C01845=1107.391,-76.844,-48.334,179.809,5.028,148.918
C01846=1107.386,-76.593,-48.345,179.809,5.034,148.919
C01847=1107.380,-76.344,-48.356,179.809,5.039,148.920
C01848=1107.375,-76.094,-48.367,179.809,5.044,148.922
C01849=1107.370,-75.844,-48.378,179.809,5.049,148.923
C01850=1107.365,-75.595,-48.389,179.809,5.054,148.924
C01851=1107.359,-75.345,-48.401,179.808,5.059,148.925
C01852=1107.354,-75.095,-48.411,179.808,5.064,148.926
C01853=1107.349,-74.846,-48.422,179.808,5.070,148.927
C01854=1107.344,-74.596,-48.434,179.808,5.075,148.929
C01855=1107.339,-74.346,-48.445,179.808,5.080,148.930
C01856=1107.333,-74.097,-48.456,179.808,5.085,148.931
C01857=1107.328,-73.847,-48.467,179.808,5.090,148.932
C01858=1107.323,-73.597,-48.478,179.807,5.095,148.933
C01859=1107.318,-73.383,-48.488,179.807,5.099,148.934
C01860=1107.314,-73.168,-48.497,179.808,5.104,148.935
C01861=1107.309,-72.954,-48.507,179.807,5.108,148.936
C01862=1107.305,-72.739,-48.517,179.808,5.113,148.937
C01863=1107.300,-72.525,-48.526,179.807,5.117,148.938
C01864=1107.296,-72.310,-48.536,179.807,5.122,148.939
C01865=1107.292,-72.096,-48.545,179.807,5.126,148.940
C01866=1107.287,-71.881,-48.555,179.807,5.131,148.941
C01867=1107.282,-71.631,-48.567,179.807,5.136,148.942
C01868=1107.276,-71.382,-48.578,179.807,5.141,148.943
C01869=1107.272,-71.132,-48.589,179.807,5.146,148.945
C01870=1107.266,-70.882,-48.601,179.807,5.151,148.946
C01871=1107.261,-70.632,-48.611,179.807,5.156,148.947
C01872=1107.255,-70.383,-48.623,179.807,5.161,148.948
C01873=1107.250,-70.133,-48.634,179.807,5.166,148.949
C01874=1107.246,-69.884,-48.645,179.807,5.171,148.950
C01875=1107.240,-69.634,-48.657,179.807,5.176,148.951
C01876=1107.235,-69.385,-48.668,179.807,5.181,148.952
C01877=1107.230,-69.135,-48.680,179.807,5.186,148.953
C01878=1107.225,-68.885,-48.691,179.807,5.191,148.955
C01879=1107.219,-68.635,-48.703,179.807,5.197,148.956
C01880=1107.214,-68.386,-48.713,179.807,5.201,148.957
C01881=1107.208,-68.136,-48.725,179.807,5.206,148.958
C01882=1107.204,-67.886,-48.737,179.807,5.212,148.959
C01883=1107.198,-67.636,-48.749,179.807,5.217,148.960
C01884=1107.194,-67.387,-48.760,179.808,5.222,148.961
C01885=1107.188,-67.137,-48.771,179.808,5.227,148.962
C01886=1107.183,-66.888,-48.783,179.807,5.233,148.963
C01887=1107.177,-66.638,-48.795,179.808,5.237,148.964
C01888=1107.173,-66.388,-48.806,179.808,5.242,148.966
C01889=1107.167,-66.138,-48.818,179.808,5.248,148.967
C01890=1107.163,-65.889,-48.829,179.808,5.252,148.968
C01891=1107.157,-65.639,-48.841,179.808,5.257,148.969
C01892=1107.152,-65.390,-48.852,179.808,5.262,148.970
C01893=1107.146,-65.140,-48.864,179.808,5.267,148.971
C01894=1107.142,-64.890,-48.875,179.809,5.273,148.972
C01895=1107.136,-64.640,-48.887,179.809,5.278,148.973
C01896=1107.132,-64.391,-48.898,179.809,5.283,148.974
C01897=1107.126,-64.141,-48.910,179.809,5.288,148.975
C01898=1107.120,-63.892,-48.922,179.809,5.293,148.976
C01899=1107.115,-63.642,-48.933,179.809,5.298,148.977
C01900=1107.110,-63.392,-48.945,179.809,5.303,148.978
C01901=1107.105,-63.142,-48.956,179.810,5.308,148.979
C01902=1107.100,-62.892,-48.968,179.810,5.313,148.980
C01903=1107.095,-62.643,-48.979,179.810,5.318,148.981
C01904=1107.090,-62.393,-48.991,179.810,5.322,148.982
C01905=1107.084,-62.144,-49.003,179.811,5.328,148.983
C01906=1107.079,-61.894,-49.014,179.811,5.333,148.984
C01907=1107.074,-61.645,-49.026,179.811,5.338,148.985
C01908=1107.069,-61.395,-49.038,179.812,5.343,148.986
C01909=1107.064,-61.145,-49.050,179.812,5.348,148.987
C01910=1107.058,-60.895,-49.062,179.812,5.353,148.988
C01911=1107.053,-60.645,-49.073,179.812,5.358,148.989
C01912=1107.048,-60.396,-49.085,179.813,5.362,148.990
C01913=1107.043,-60.146,-49.097,179.812,5.367,148.992
C01914=1107.038,-59.896,-49.109,179.813,5.372,148.992
C01915=1107.033,-59.682,-49.119,179.813,5.377,148.993
C01916=1107.029,-59.468,-49.130,179.813,5.381,148.994
C01917=1107.024,-59.253,-49.140,179.813,5.385,148.995
C01918=1107.020,-59.038,-49.150,179.813,5.389,148.996
C01919=1107.015,-58.825,-49.160,179.812,5.393,148.997
C01920=1107.011,-58.610,-49.170,179.812,5.397,148.998
C01921=1107.007,-58.395,-49.180,179.812,5.401,148.999
C01922=1107.002,-58.181,-49.190,179.813,5.405,149.000
C01923=1106.997,-57.931,-49.202,179.812,5.409,149.001
C01924=1106.992,-57.682,-49.213,179.812,5.414,149.002
C01925=1106.987,-57.433,-49.226,179.812,5.418,149.003
C01926=1106.981,-57.183,-49.238,179.812,5.423,149.004
C01927=1106.977,-56.933,-49.249,179.812,5.428,149.005
C01928=1106.971,-56.683,-49.261,179.812,5.433,149.006
C01929=1106.966,-56.434,-49.274,179.811,5.438,149.007
C01930=1106.961,-56.184,-49.286,179.812,5.442,149.008
C01931=1106.956,-55.934,-49.297,179.811,5.447,149.009
C01932=1106.951,-55.685,-49.310,179.811,5.452,149.010
C01933=1106.946,-55.435,-49.321,179.812,5.457,149.011
C01934=1106.940,-55.185,-49.333,179.811,5.461,149.013
C01935=1106.935,-54.936,-49.346,179.811,5.466,149.013
C01936=1106.930,-54.686,-49.357,179.811,5.471,149.015
C01937=1106.925,-54.437,-49.370,179.810,5.475,149.016
C01938=1106.920,-54.187,-49.382,179.811,5.480,149.017
C01939=1106.914,-53.937,-49.394,179.811,5.485,149.018
C01940=1106.909,-53.688,-49.406,179.810,5.489,149.019
C01941=1106.905,-53.438,-49.417,179.810,5.494,149.020
C01942=1106.900,-53.187,-49.430,179.810,5.499,149.021
C01943=1106.895,-52.938,-49.442,179.810,5.504,149.022
C01944=1106.889,-52.688,-49.454,179.810,5.508,149.023
C01945=1106.884,-52.439,-49.467,179.809,5.513,149.024
C01946=1106.879,-52.189,-49.479,179.809,5.518,149.025
C01947=1106.874,-51.940,-49.491,179.810,5.522,149.026
C01948=1106.869,-51.690,-49.503,179.809,5.527,149.028
C01949=1106.864,-51.440,-49.515,179.809,5.532,149.029
C01950=1106.858,-51.191,-49.527,179.809,5.537,149.030
C01951=1106.853,-50.941,-49.539,179.809,5.541,149.031
C01952=1106.848,-50.691,-49.552,179.809,5.546,149.032
C01953=1106.842,-50.441,-49.563,179.809,5.551,149.033
C01954=1106.837,-50.192,-49.576,179.808,5.555,149.034
C01955=1106.832,-49.942,-49.588,179.808,5.560,149.035
C01956=1106.827,-49.693,-49.600,179.809,5.565,149.036
C01957=1106.822,-49.444,-49.612,179.808,5.569,149.037
C01958=1106.817,-49.193,-49.625,179.808,5.574,149.038
C01959=1106.812,-48.944,-49.637,179.808,5.578,149.039
C01960=1106.807,-48.694,-49.649,179.808,5.584,149.040
C01961=1106.802,-48.445,-49.662,179.808,5.589,149.042
C01962=1106.796,-48.195,-49.674,179.807,5.593,149.043
C01963=1106.791,-47.945,-49.686,179.807,5.598,149.044
C01964=1106.786,-47.695,-49.698,179.807,5.603,149.045
C01965=1106.781,-47.446,-49.711,179.807,5.607,149.046
C01966=1106.775,-47.197,-49.723,179.807,5.612,149.047
C01967=1106.770,-46.947,-49.735,179.807,5.617,149.048
C01968=1106.765,-46.697,-49.748,179.806,5.621,149.049
C01969=1106.760,-46.447,-49.760,179.806,5.627,149.050
C01970=1106.755,-46.198,-49.773,179.806,5.630,149.051
C01971=1106.751,-45.983,-49.783,179.807,5.635,149.052
C01972=1106.747,-45.768,-49.793,179.806,5.639,149.053
C01973=1106.741,-45.555,-49.804,179.806,5.643,149.054
C01974=1106.737,-45.340,-49.815,179.806,5.647,149.055
C01975=1106.733,-45.126,-49.826,179.805,5.651,149.056
C01976=1106.729,-44.911,-49.836,179.805,5.655,149.057
C01977=1106.724,-44.697,-49.847,179.805,5.659,149.058
C01978=1106.720,-44.482,-49.858,179.805,5.663,149.059
C01979=1106.715,-44.233,-49.871,179.805,5.668,149.060
C01980=1106.709,-43.983,-49.882,179.805,5.673,149.061
C01981=1106.704,-43.734,-49.895,179.805,5.677,149.062
C01982=1106.699,-43.485,-49.908,179.805,5.682,149.063
C01983=1106.694,-43.235,-49.920,179.804,5.686,149.064
C01984=1106.689,-42.985,-49.932,179.804,5.692,149.065
C01985=1106.684,-42.735,-49.945,179.804,5.697,149.066
C01986=1106.679,-42.486,-49.958,179.805,5.701,149.067
C01987=1106.674,-42.236,-49.970,179.805,5.706,149.068
C01988=1106.668,-41.986,-49.983,179.805,5.711,149.069
C01989=1106.663,-41.736,-49.996,179.806,5.716,149.070
C01990=1106.658,-41.487,-50.008,179.806,5.721,149.071
C01991=1106.653,-41.238,-50.021,179.806,5.726,149.072
C01992=1106.647,-40.988,-50.033,179.806,5.731,149.073
C01993=1106.642,-40.739,-50.045,179.807,5.735,149.074
C01994=1106.638,-40.488,-50.058,179.807,5.740,149.075
C01995=1106.633,-40.239,-50.071,179.808,5.745,149.076
C01996=1106.628,-39.990,-50.084,179.808,5.750,149.077
C01997=1106.621,-39.740,-50.096,179.808,5.755,149.078
C01998=1106.617,-39.490,-50.109,179.809,5.759,149.079
C01999=1106.612,-39.240,-50.122,179.809,5.764,149.080
C02000=1106.607,-38.991,-50.134,179.809,5.769,149.081
C02001=1106.602,-38.742,-50.147,179.810,5.774,149.082
C02002=1106.597,-38.492,-50.160,179.810,5.778,149.083
C02003=1106.591,-38.242,-50.173,179.811,5.783,149.084
C02004=1106.586,-37.993,-50.186,179.811,5.788,149.084
C02005=1106.581,-37.743,-50.197,179.811,5.792,149.085
C02006=1106.576,-37.493,-50.210,179.811,5.796,149.086
C02007=1106.571,-37.243,-50.223,179.812,5.801,149.087
C02008=1106.565,-36.994,-50.236,179.812,5.806,149.088
C02009=1106.560,-36.744,-50.249,179.813,5.811,149.089
C02010=1106.555,-36.494,-50.262,179.814,5.815,149.090
C02011=1106.550,-36.245,-50.274,179.814,5.819,149.091
C02012=1106.544,-35.995,-50.288,179.814,5.824,149.091
C02013=1106.540,-35.745,-50.301,179.815,5.828,149.092
C02014=1106.535,-35.496,-50.313,179.815,5.833,149.093
C02015=1106.530,-35.247,-50.326,179.815,5.837,149.094
C02016=1106.524,-34.996,-50.339,179.815,5.842,149.095
C02017=1106.519,-34.747,-50.352,179.816,5.847,149.096
C02018=1106.514,-34.498,-50.364,179.816,5.851,149.097
C02019=1106.510,-34.248,-50.377,179.816,5.855,149.098
C02020=1106.504,-33.998,-50.391,179.817,5.860,149.099
C02021=1106.499,-33.749,-50.403,179.817,5.864,149.099
C02022=1106.494,-33.499,-50.416,179.817,5.868,149.100
C02023=1106.488,-33.249,-50.429,179.818,5.873,149.101
C02024=1106.483,-33.000,-50.442,179.818,5.878,149.102
C02025=1106.479,-32.750,-50.455,179.819,5.882,149.103
C02026=1106.474,-32.501,-50.468,179.818,5.886,149.104
C02027=1106.469,-32.287,-50.480,179.819,5.890,149.105
C02028=1106.464,-32.072,-50.491,179.820,5.894,149.105
C02029=1106.460,-31.858,-50.502,179.820,5.898,149.106
C02030=1106.455,-31.643,-50.513,179.820,5.902,149.107
C02031=1106.452,-31.430,-50.524,179.820,5.906,149.108
C02032=1106.447,-31.215,-50.536,179.820,5.909,149.109
C02033=1106.443,-31.001,-50.546,179.821,5.913,149.109
C02034=1106.438,-30.786,-50.558,179.820,5.917,149.110
C02035=1106.433,-30.537,-50.570,179.821,5.921,149.111
C02036=1106.428,-30.287,-50.584,179.821,5.926,149.112
C02037=1106.423,-30.038,-50.597,179.821,5.930,149.113
C02038=1106.418,-29.788,-50.610,179.822,5.935,149.114
C02039=1106.413,-29.538,-50.623,179.822,5.940,149.115
C02040=1106.407,-29.289,-50.636,179.822,5.944,149.116
C02041=1106.402,-29.039,-50.650,179.822,5.948,149.116
C02042=1106.397,-28.790,-50.663,179.822,5.952,149.117
C02043=1106.393,-28.540,-50.676,179.823,5.957,149.118
C02044=1106.387,-28.290,-50.689,179.823,5.962,149.119
C02045=1106.382,-28.041,-50.702,179.823,5.966,149.120
C02046=1106.377,-27.791,-50.716,179.824,5.970,149.121
C02047=1106.372,-27.542,-50.729,179.824,5.975,149.122
C02048=1106.367,-27.292,-50.741,179.823,5.979,149.123
C02049=1106.361,-27.042,-50.755,179.824,5.984,149.124
C02050=1106.357,-26.793,-50.768,179.824,5.989,149.125
C02051=1106.351,-26.543,-50.782,179.824,5.993,149.126
C02052=1106.347,-26.293,-50.795,179.824,5.998,149.127
C02053=1106.341,-26.044,-50.808,179.824,6.002,149.128
C02054=1106.337,-25.794,-50.821,179.825,6.007,149.129
C02055=1106.331,-25.545,-50.835,179.824,6.012,149.130
C02056=1106.327,-25.295,-50.848,179.825,6.016,149.131
C02057=1106.321,-25.046,-50.861,179.825,6.021,149.132
C02058=1106.316,-24.796,-50.874,179.825,6.025,149.133
C02059=1106.311,-24.547,-50.888,179.826,6.030,149.133
C02060=1106.306,-24.297,-50.901,179.826,6.035,149.135
C02061=1106.300,-24.047,-50.915,179.826,6.040,149.136
C02062=1106.296,-23.798,-50.928,179.827,6.044,149.136
C02063=1106.290,-23.548,-50.941,179.827,6.049,149.137
C02064=1106.285,-23.299,-50.955,179.828,6.054,149.138
C02065=1106.280,-23.049,-50.968,179.828,6.058,149.139
C02066=1106.275,-22.800,-50.981,179.828,6.063,149.140
C02067=1106.270,-22.550,-50.995,179.828,6.068,149.141
C02068=1106.264,-22.300,-51.008,179.829,6.072,149.142
C02069=1106.260,-22.051,-51.022,179.829,6.077,149.143
C02070=1106.254,-21.801,-51.035,179.829,6.082,149.144
C02071=1106.250,-21.552,-51.049,179.830,6.086,149.145
C02072=1106.245,-21.302,-51.062,179.830,6.091,149.146
C02073=1106.240,-21.053,-51.076,179.830,6.095,149.147
C02074=1106.235,-20.802,-51.089,179.831,6.100,149.147
C02075=1106.229,-20.553,-51.103,179.831,6.105,149.148
C02076=1106.225,-20.303,-51.116,179.832,6.109,149.149
C02077=1106.219,-20.054,-51.130,179.832,6.114,149.150
C02078=1106.214,-19.804,-51.144,179.833,6.119,149.151
C02079=1106.209,-19.555,-51.157,179.833,6.123,149.152
C02080=1106.204,-19.305,-51.171,179.833,6.127,149.153
C02081=1106.199,-19.056,-51.184,179.834,6.132,149.154
C02082=1106.194,-18.806,-51.197,179.834,6.137,149.155
C02083=1106.189,-18.592,-51.209,179.834,6.141,149.156
C02084=1106.185,-18.378,-51.222,179.835,6.145,149.156
C02085=1106.180,-18.163,-51.233,179.835,6.149,149.157
C02086=1106.177,-17.949,-51.245,179.835,6.153,149.158
C02087=1106.172,-17.735,-51.256,179.836,6.157,149.159
C02088=1106.168,-17.521,-51.268,179.836,6.161,149.159
C02089=1106.163,-17.307,-51.280,179.836,6.164,149.160
C02090=1106.158,-17.092,-51.291,179.837,6.168,149.161
C02091=1106.154,-16.843,-51.305,179.837,6.173,149.162
C02092=1106.149,-16.594,-51.319,179.838,6.177,149.163
C02093=1106.143,-16.344,-51.332,179.838,6.182,149.163
C02094=1106.138,-16.094,-51.347,179.839,6.187,149.164
C02095=1106.133,-15.845,-51.360,179.839,6.192,149.165
C02096=1106.128,-15.595,-51.374,179.839,6.195,149.166
C02097=1106.123,-15.345,-51.388,179.840,6.200,149.167
C02098=1106.118,-15.096,-51.401,179.840,6.205,149.168
C02099=1106.113,-14.846,-51.415,179.841,6.209,149.169
C02100=1106.108,-14.596,-51.429,179.842,6.214,149.170
C02101=1106.103,-14.347,-51.443,179.842,6.219,149.170
C02102=1106.098,-14.098,-51.457,179.843,6.223,149.171
C02103=1106.093,-13.848,-51.470,179.842,6.227,149.172
C02104=1106.088,-13.599,-51.484,179.843,6.232,149.173
C02105=1106.083,-13.349,-51.498,179.843,6.237,149.174
C02106=1106.078,-13.099,-51.513,179.844,6.241,149.175
C02107=1106.073,-12.850,-51.525,179.845,6.246,149.176
C02108=1106.068,-12.600,-51.540,179.845,6.251,149.176
C02109=1106.063,-12.351,-51.554,179.845,6.254,149.177
C02110=1106.057,-12.102,-51.568,179.846,6.259,149.178
C02111=1106.052,-11.852,-51.582,179.847,6.264,149.179
C02112=1106.047,-11.602,-51.596,179.847,6.268,149.180
C02113=1106.043,-11.352,-51.609,179.848,6.273,149.181
C02114=1106.037,-11.103,-51.623,179.848,6.278,149.182
C02115=1106.032,-10.853,-51.637,179.849,6.282,149.183
C02116=1106.027,-10.604,-51.652,179.849,6.286,149.183
C02117=1106.022,-10.355,-51.666,179.850,6.291,149.184
C02118=1106.017,-10.105,-51.680,179.850,6.295,149.185
C02119=1106.013,-9.856,-51.694,179.851,6.300,149.186
C02120=1106.008,-9.606,-51.708,179.851,6.305,149.187
C02121=1106.002,-9.356,-51.721,179.852,6.309,149.187
C02122=1105.997,-9.106,-51.735,179.853,6.314,149.188
C02123=1105.992,-8.857,-51.750,179.853,6.318,149.189
C02124=1105.987,-8.607,-51.764,179.853,6.322,149.190
C02125=1105.981,-8.358,-51.778,179.854,6.327,149.191
C02126=1105.976,-8.108,-51.792,179.855,6.332,149.192
C02127=1105.971,-7.859,-51.806,179.855,6.336,149.193
C02128=1105.966,-7.609,-51.821,179.856,6.341,149.194
C02129=1105.961,-7.359,-51.835,179.857,6.345,149.194
C02130=1105.956,-7.110,-51.849,179.857,6.349,149.195
C02131=1105.951,-6.860,-51.863,179.857,6.354,149.196
C02132=1105.947,-6.611,-51.877,179.858,6.359,149.197
C02133=1105.942,-6.361,-51.891,179.859,6.363,149.198
C02134=1105.937,-6.112,-51.905,179.859,6.368,149.198
C02135=1105.931,-5.863,-51.919,179.860,6.372,149.199
C02136=1105.926,-5.613,-51.934,179.861,6.377,149.200
C02137=1105.921,-5.363,-51.948,179.861,6.381,149.201
C02138=1105.916,-5.114,-51.962,179.861,6.385,149.202
C02139=1105.912,-4.900,-51.974,179.862,6.390,149.202
C02140=1105.907,-4.686,-51.987,179.862,6.393,149.203
C02141=1105.903,-4.471,-52.000,179.863,6.397,149.204
C02142=1105.899,-4.257,-52.012,179.863,6.402,149.205
C02143=1105.894,-4.044,-52.024,179.864,6.405,149.205
C02144=1105.890,-3.829,-52.036,179.864,6.409,149.206
C02145=1105.886,-3.615,-52.048,179.865,6.413,149.207
C02146=1105.881,-3.401,-52.060,179.865,6.416,149.207
C02147=1105.877,-3.151,-52.075,179.866,6.421,149.208
C02148=1105.872,-2.902,-52.089,179.867,6.426,149.209
C02149=1105.867,-2.653,-52.104,179.867,6.431,149.210
C02150=1105.861,-2.402,-52.119,179.868,6.435,149.211
C02151=1105.856,-2.153,-52.133,179.869,6.440,149.212
C02152=1105.851,-1.904,-52.147,179.869,6.444,149.212
C02153=1105.846,-1.654,-52.161,179.869,6.448,149.213
C02154=1105.841,-1.405,-52.176,179.870,6.453,149.214
C02155=1105.836,-1.155,-52.191,179.871,6.457,149.215
C02156=1105.831,-0.906,-52.205,179.871,6.462,149.216
C02157=1105.826,-0.656,-52.219,179.872,6.466,149.217
C02158=1105.821,-0.406,-52.233,179.873,6.471,149.217
C02159=1105.816,-0.157,-52.249,179.873,6.476,149.218
C02160=1105.811,0.093,-52.263,179.874,6.480,149.219
C02161=1105.805,0.342,-52.277,179.875,6.485,149.220
C02162=1105.801,0.591,-52.292,179.875,6.490,149.221
C02163=1105.796,0.841,-52.306,179.876,6.494,149.221
C02164=1105.791,1.091,-52.321,179.877,6.499,149.222
C02165=1105.786,1.340,-52.335,179.877,6.503,149.223
C02166=1105.780,1.590,-52.351,179.878,6.508,149.224
C02167=1105.776,1.839,-52.365,179.878,6.512,149.225
C02168=1105.771,2.089,-52.379,179.879,6.516,149.226
C02169=1105.766,2.338,-52.394,179.879,6.521,149.227
C02170=1105.761,2.588,-52.408,179.880,6.525,149.227
C02171=1105.756,2.837,-52.424,179.881,6.530,149.228
C02172=1105.751,3.087,-52.438,179.881,6.535,149.229
C02173=1105.746,3.337,-52.453,179.882,6.539,149.230
C02174=1105.741,3.586,-52.468,179.883,6.544,149.231
C02175=1105.735,3.836,-52.482,179.883,6.548,149.231
C02176=1105.731,4.085,-52.497,179.884,6.553,149.232
C02177=1105.726,4.335,-52.512,179.884,6.558,149.233
C02178=1105.721,4.584,-52.526,179.885,6.562,149.234
C02179=1105.715,4.834,-52.542,179.886,6.567,149.235
C02180=1105.710,5.083,-52.556,179.887,6.572,149.236
C02181=1105.706,5.333,-52.571,179.887,6.576,149.237
C02182=1105.701,5.582,-52.585,179.888,6.581,149.237
C02183=1105.695,5.832,-52.601,179.889,6.585,149.238
C02184=1105.690,6.081,-52.615,179.889,6.590,149.239
C02185=1105.686,6.330,-52.630,179.890,6.595,149.240
C02186=1105.680,6.580,-52.645,179.891,6.599,149.241
C02187=1105.675,6.830,-52.660,179.891,6.604,149.241
C02188=1105.671,7.079,-52.674,179.892,6.608,149.242
C02189=1105.665,7.329,-52.690,179.892,6.613,149.243
C02190=1105.661,7.578,-52.705,179.893,6.618,149.244
C02191=1105.656,7.827,-52.719,179.894,6.622,149.245
C02192=1105.650,8.077,-52.735,179.894,6.627,149.246
C02193=1105.645,8.327,-52.749,179.895,6.632,149.247
C02194=1105.641,8.576,-52.764,179.896,6.636,149.247
C02195=1105.636,8.791,-52.777,179.896,6.640,149.248
C02196=1105.632,9.004,-52.790,179.897,6.644,149.249
C02197=1105.628,9.218,-52.803,179.897,6.648,149.250
C02198=1105.623,9.432,-52.815,179.897,6.652,149.250
C02199=1105.619,9.646,-52.828,179.897,6.656,149.251
C02200=1105.614,9.860,-52.841,179.898,6.659,149.252
C02201=1105.611,10.074,-52.854,179.899,6.663,149.253
C02202=1105.606,10.288,-52.867,179.899,6.667,149.253
C02203=1105.601,10.538,-52.882,179.899,6.671,149.254
C02204=1105.595,10.787,-52.897,179.899,6.676,149.255
C02205=1105.591,11.036,-52.912,179.900,6.681,149.256
C02206=1105.586,11.286,-52.927,179.901,6.685,149.257
C02207=1105.581,11.536,-52.943,179.901,6.689,149.258
C02208=1105.576,11.785,-52.958,179.901,6.694,149.259
C02209=1105.571,12.035,-52.972,179.902,6.698,149.259
C02210=1105.566,12.284,-52.987,179.902,6.702,149.260
C02211=1105.561,12.534,-53.003,179.902,6.707,149.261
C02212=1105.556,12.783,-53.018,179.903,6.712,149.262
C02213=1105.550,13.033,-53.033,179.903,6.716,149.263
C02214=1105.546,13.282,-53.048,179.904,6.720,149.264
C02215=1105.541,13.532,-53.064,179.904,6.725,149.264
C02216=1105.536,13.781,-53.079,179.905,6.729,149.265
C02217=1105.531,14.031,-53.094,179.905,6.733,149.266
C02218=1105.526,14.280,-53.109,179.905,6.738,149.267
C02219=1105.521,14.530,-53.124,179.906,6.742,149.268
C02220=1105.516,14.779,-53.139,179.907,6.747,149.269
C02221=1105.511,15.029,-53.155,179.907,6.751,149.270
C02222=1105.506,15.278,-53.170,179.907,6.755,149.270
C02223=1105.501,15.528,-53.185,179.909,6.760,149.271
C02224=1105.496,15.777,-53.200,179.908,6.764,149.272
C02225=1105.491,16.026,-53.216,179.909,6.768,149.273
C02226=1105.487,16.276,-53.231,179.910,6.773,149.274
C02227=1105.481,16.526,-53.247,179.910,6.777,149.274
C02228=1105.476,16.775,-53.262,179.911,6.781,149.275
C02229=1105.471,17.024,-53.277,179.911,6.786,149.276
C02230=1105.466,17.273,-53.293,179.912,6.790,149.277
C02231=1105.462,17.524,-53.307,179.912,6.794,149.278
C02232=1105.456,17.773,-53.323,179.913,6.799,149.279
C02233=1105.451,18.023,-53.339,179.914,6.803,149.279
C02234=1105.446,18.272,-53.354,179.914,6.807,149.280
C02235=1105.441,18.521,-53.369,179.914,6.812,149.281
C02236=1105.437,18.771,-53.385,179.915,6.816,149.282
C02237=1105.431,19.020,-53.400,179.915,6.820,149.283
C02238=1105.426,19.270,-53.416,179.916,6.824,149.283
C02239=1105.421,19.519,-53.431,179.917,6.829,149.284
C02240=1105.416,19.769,-53.447,179.917,6.833,149.285
C02241=1105.411,20.018,-53.462,179.918,6.837,149.286
C02242=1105.406,20.267,-53.477,179.918,6.842,149.287
C02243=1105.401,20.517,-53.493,179.919,6.846,149.287
C02244=1105.396,20.767,-53.509,179.919,6.850,149.288
C02245=1105.392,21.016,-53.524,179.920,6.855,149.289
C02246=1105.386,21.265,-53.539,179.921,6.859,149.290
C02247=1105.381,21.516,-53.555,179.921,6.863,149.290
C02248=1105.377,21.765,-53.570,179.922,6.868,149.291
C02249=1105.371,22.014,-53.586,179.923,6.872,149.292
C02250=1105.366,22.263,-53.602,179.923,6.876,149.293
C02251=1105.362,22.477,-53.616,179.924,6.880,149.293
C02252=1105.358,22.691,-53.629,179.925,6.884,149.294
C02253=1105.354,22.905,-53.642,179.925,6.887,149.295
C02254=1105.349,23.119,-53.656,179.925,6.891,149.295
C02255=1105.346,23.333,-53.669,179.926,6.894,149.296
C02256=1105.341,23.547,-53.683,179.926,6.898,149.297
C02257=1105.337,23.761,-53.696,179.927,6.902,149.297
C02258=1105.332,23.974,-53.709,179.928,6.905,149.298
C02259=1105.328,24.224,-53.725,179.928,6.909,149.299
C02260=1105.322,24.474,-53.741,179.929,6.914,149.300
C02261=1105.317,24.723,-53.756,179.930,6.918,149.300
C02262=1105.313,24.972,-53.772,179.930,6.922,149.301
C02263=1105.308,25.222,-53.788,179.931,6.926,149.302
C02264=1105.302,25.471,-53.803,179.932,6.931,149.302
C02265=1105.298,25.721,-53.819,179.932,6.935,149.303
C02266=1105.292,25.971,-53.835,179.933,6.939,149.304
C02267=1105.288,26.219,-53.851,179.934,6.943,149.305
C02268=1105.283,26.469,-53.867,179.934,6.948,149.306
C02269=1105.278,26.719,-53.882,179.935,6.951,149.306
C02270=1105.273,26.969,-53.898,179.936,6.956,149.307
C02271=1105.268,27.218,-53.914,179.937,6.960,149.308
C02272=1105.262,27.467,-53.930,179.937,6.964,149.308
C02273=1105.258,27.717,-53.945,179.938,6.968,149.309
C02274=1105.253,27.966,-53.961,179.939,6.973,149.310
C02275=1105.248,28.215,-53.977,179.939,6.976,149.311
C02276=1105.243,28.465,-53.993,179.940,6.981,149.311
C02277=1105.238,28.715,-54.009,179.941,6.985,149.312
C02278=1105.233,28.964,-54.025,179.942,6.990,149.313
C02279=1105.228,29.213,-54.041,179.942,6.993,149.313
C02280=1105.223,29.464,-54.057,179.943,6.997,149.314
C02281=1105.219,29.712,-54.073,179.944,7.002,149.315
C02282=1105.213,29.961,-54.088,179.944,7.006,149.316
C02283=1105.209,30.211,-54.105,179.945,7.010,149.316
C02284=1105.203,30.460,-54.121,179.946,7.014,149.317
C02285=1105.199,30.710,-54.136,179.946,7.018,149.318
C02286=1105.194,30.959,-54.153,179.947,7.023,149.318
C02287=1105.189,31.209,-54.169,179.949,7.027,149.319
C02288=1105.184,31.458,-54.185,179.949,7.030,149.320
C02289=1105.178,31.707,-54.201,179.950,7.035,149.320
C02290=1105.174,31.958,-54.217,179.951,7.039,149.321
C02291=1105.168,32.206,-54.233,179.952,7.044,149.322
C02292=1105.164,32.456,-54.249,179.952,7.047,149.323
C02293=1105.159,32.705,-54.265,179.953,7.051,149.323
C02294=1105.154,32.955,-54.281,179.954,7.056,149.324
C02295=1105.149,33.204,-54.297,179.955,7.059,149.325
C02296=1105.144,33.454,-54.313,179.956,7.064,149.325
C02297=1105.139,33.703,-54.330,179.956,7.068,149.326
C02298=1105.134,33.953,-54.346,179.957,7.072,149.327
C02299=1105.129,34.202,-54.362,179.958,7.076,149.327
C02300=1105.124,34.452,-54.378,179.959,7.080,149.328
C02301=1105.119,34.701,-54.394,179.959,7.084,149.329
C02302=1105.114,34.951,-54.410,179.960,7.088,149.329
C02303=1105.109,35.200,-54.426,179.961,7.093,149.330
C02304=1105.105,35.449,-54.443,179.963,7.097,149.331
C02305=1105.099,35.699,-54.459,179.963,7.100,149.331
C02306=1105.095,35.948,-54.475,179.964,7.105,149.332
C02307=1105.090,36.162,-54.489,179.965,7.108,149.333
C02308=1105.086,36.375,-54.503,179.965,7.112,149.333
C02309=1105.082,36.590,-54.517,179.966,7.115,149.334
C02310=1105.078,36.803,-54.531,179.967,7.119,149.334
C02311=1105.073,37.018,-54.545,179.967,7.123,149.335
C02312=1105.069,37.231,-54.559,179.968,7.126,149.336
C02313=1105.065,37.445,-54.573,179.969,7.129,149.336
C02314=1105.061,37.659,-54.587,179.970,7.132,149.337
C02315=1105.056,37.908,-54.604,179.971,7.137,149.337
C02316=1105.051,38.158,-54.619,179.972,7.141,149.338
C02317=1105.046,38.407,-54.636,179.972,7.145,149.339
C02318=1105.040,38.656,-54.653,179.973,7.149,149.339
C02319=1105.036,38.906,-54.669,179.974,7.153,149.340
C02320=1105.031,39.155,-54.685,179.975,7.157,149.341
C02321=1105.026,39.405,-54.702,179.976,7.161,149.341
C02322=1105.021,39.655,-54.718,179.977,7.165,149.342
C02323=1105.016,39.903,-54.734,179.978,7.170,149.343
C02324=1105.011,40.153,-54.751,179.979,7.173,149.343
C02325=1105.006,40.402,-54.768,179.980,7.177,149.344
C02326=1105.001,40.651,-54.784,179.981,7.182,149.345
C02327=1104.997,40.902,-54.800,179.982,7.186,149.345
C02328=1104.992,41.150,-54.817,179.982,7.190,149.346
C02329=1104.986,41.400,-54.834,179.983,7.194,149.346
C02330=1104.981,41.649,-54.850,179.984,7.198,149.347
C02331=1104.977,41.898,-54.867,179.985,7.202,149.348
C02332=1104.972,42.149,-54.883,179.986,7.206,149.348
C02333=1104.967,42.397,-54.899,179.987,7.210,149.349
C02334=1104.962,42.647,-54.916,179.988,7.213,149.350
C02335=1104.957,42.897,-54.933,179.989,7.218,149.350
C02336=1104.952,43.145,-54.949,179.990,7.222,149.351
C02337=1104.948,43.395,-54.966,179.991,7.226,149.352
C02338=1104.942,43.645,-54.983,179.992,7.230,149.352
C02339=1104.937,43.894,-54.999,179.993,7.234,149.353
C02340=1104.933,44.144,-55.016,179.994,7.238,149.353
C02341=1104.927,44.393,-55.033,179.995,7.242,149.354
C02342=1104.922,44.642,-55.049,179.996,7.246,149.355
C02343=1104.918,44.892,-55.066,179.997,7.250,149.355
C02344=1104.913,45.141,-55.083,179.998,7.254,149.356
C02345=1104.907,45.390,-55.099,179.998,7.258,149.357
C02346=1104.903,45.640,-55.116,180.000,7.262,149.357
C02347=1104.899,45.889,-55.133,-179.999,7.266,149.358
C02348=1104.893,46.138,-55.150,-179.998,7.270,149.358
C02349=1104.888,46.388,-55.166,-179.997,7.274,149.359
C02350=1104.883,46.638,-55.184,-179.996,7.278,149.360
C02351=1104.879,46.887,-55.200,-179.995,7.282,149.360
C02352=1104.873,47.136,-55.217,-179.994,7.286,149.361
C02353=1104.868,47.386,-55.234,-179.993,7.290,149.361
C02354=1104.864,47.635,-55.250,-179.992,7.294,149.362
C02355=1104.859,47.885,-55.267,-179.991,7.298,149.362
C02356=1104.853,48.134,-55.284,-179.990,7.302,149.363
C02357=1104.849,48.383,-55.301,-179.989,7.306,149.364
C02358=1104.844,48.633,-55.318,-179.988,7.310,149.364
C02359=1104.840,48.882,-55.335,-179.986,7.314,149.365
C02360=1104.835,49.131,-55.352,-179.986,7.318,149.365
C02361=1104.829,49.380,-55.369,-179.985,7.322,149.366
C02362=1104.825,49.630,-55.386,-179.983,7.326,149.367
C02363=1104.821,49.844,-55.400,-179.983,7.329,149.367
C02364=1104.816,50.058,-55.415,-179.982,7.333,149.368
C02365=1104.812,50.271,-55.429,-179.981,7.336,149.368
C02366=1104.808,50.485,-55.444,-179.980,7.340,149.369
C02367=1104.804,50.699,-55.458,-179.979,7.343,149.369
C02368=1104.799,50.913,-55.473,-179.978,7.346,149.370
C02369=1104.795,51.126,-55.488,-179.978,7.350,149.370
C02370=1104.791,51.340,-55.502,-179.977,7.353,149.371
C02371=1104.786,51.589,-55.519,-179.976,7.357,149.371
C02372=1104.781,51.839,-55.536,-179.974,7.361,149.372
C02373=1104.776,52.088,-55.553,-179.973,7.365,149.372
C02374=1104.772,52.337,-55.570,-179.973,7.369,149.373
C02375=1104.767,52.587,-55.588,-179.971,7.373,149.374
C02376=1104.761,52.836,-55.604,-179.970,7.377,149.374
C02377=1104.756,53.086,-55.621,-179.969,7.381,149.375
C02378=1104.752,53.335,-55.639,-179.968,7.385,149.375
C02379=1104.747,53.584,-55.656,-179.967,7.389,149.376
C02380=1104.742,53.834,-55.673,-179.965,7.393,149.376
C02381=1104.737,54.083,-55.691,-179.964,7.397,149.377
C02382=1104.732,54.332,-55.707,-179.964,7.401,149.378
C02383=1104.727,54.582,-55.724,-179.962,7.404,149.378
C02384=1104.722,54.831,-55.742,-179.961,7.409,149.379
C02385=1104.718,55.080,-55.759,-179.960,7.413,149.379
C02386=1104.713,55.330,-55.776,-179.958,7.417,149.380
C02387=1104.708,55.579,-55.794,-179.958,7.420,149.381
C02388=1104.703,55.829,-55.811,-179.956,7.424,149.381
C02389=1104.698,56.078,-55.828,-179.955,7.429,149.382
C02390=1104.693,56.327,-55.845,-179.954,7.433,149.382
C02391=1104.688,56.576,-55.862,-179.953,7.436,149.383
C02392=1104.683,56.826,-55.880,-179.952,7.440,149.383
C02393=1104.679,57.075,-55.897,-179.951,7.444,149.384
C02394=1104.673,57.325,-55.914,-179.949,7.449,149.384
C02395=1104.668,57.574,-55.932,-179.949,7.452,149.385
C02396=1104.664,57.824,-55.949,-179.947,7.456,149.386
C02397=1104.659,58.073,-55.967,-179.946,7.460,149.386
C02398=1104.654,58.323,-55.984,-179.945,7.464,149.387
C02399=1104.650,58.571,-56.001,-179.943,7.468,149.387
C02400=1104.644,58.821,-56.019,-179.943,7.472,149.388
C02401=1104.639,59.070,-56.036,-179.941,7.476,149.388
C02402=1104.634,59.319,-56.053,-179.940,7.480,149.389
C02403=1104.630,59.568,-56.071,-179.939,7.484,149.389
C02404=1104.624,59.818,-56.088,-179.938,7.487,149.390
C02405=1104.619,60.067,-56.106,-179.937,7.491,149.391
C02406=1104.615,60.317,-56.123,-179.935,7.495,149.391
C02407=1104.610,60.566,-56.141,-179.934,7.500,149.392
C02408=1104.605,60.815,-56.159,-179.933,7.504,149.392
C02409=1104.600,61.065,-56.176,-179.932,7.507,149.393
C02410=1104.596,61.314,-56.193,-179.931,7.511,149.393
C02411=1104.590,61.564,-56.211,-179.929,7.515,149.394
C02412=1104.586,61.813,-56.229,-179.928,7.519,149.394
C02413=1104.581,62.062,-56.247,-179.926,7.523,149.395
C02414=1104.576,62.311,-56.263,-179.926,7.527,149.395
C02415=1104.571,62.561,-56.281,-179.924,7.531,149.396
C02416=1104.566,62.810,-56.299,-179.923,7.535,149.396
C02417=1104.561,63.060,-56.317,-179.922,7.539,149.397
C02418=1104.556,63.309,-56.335,-179.921,7.543,149.398
C02419=1104.552,63.522,-56.349,-179.920,7.546,149.398
C02420=1104.548,63.736,-56.365,-179.919,7.549,149.398
C02421=1104.544,63.950,-56.379,-179.918,7.552,149.399
C02422=1104.540,64.164,-56.395,-179.916,7.556,149.399
C02423=1104.536,64.377,-56.410,-179.915,7.559,149.400
C02424=1104.532,64.591,-56.425,-179.914,7.563,149.400
C02425=1104.527,64.805,-56.440,-179.913,7.566,149.401
C02426=1104.523,65.018,-56.456,-179.912,7.570,149.401
C02427=1104.518,65.267,-56.473,-179.911,7.574,149.402
C02428=1104.514,65.517,-56.492,-179.910,7.577,149.402
C02429=1104.509,65.767,-56.509,-179.909,7.581,149.403
C02430=1104.504,66.016,-56.527,-179.907,7.585,149.403
C02431=1104.499,66.265,-56.545,-179.906,7.589,149.404
C02432=1104.495,66.514,-56.562,-179.904,7.593,149.404
C02433=1104.490,66.763,-56.580,-179.903,7.597,149.405
C02434=1104.485,67.013,-56.598,-179.902,7.601,149.405
C02435=1104.480,67.262,-56.616,-179.901,7.605,149.406
C02436=1104.475,67.511,-56.634,-179.900,7.609,149.406
C02437=1104.470,67.760,-56.652,-179.898,7.613,149.407
C02438=1104.465,68.010,-56.670,-179.897,7.617,149.407
C02439=1104.461,68.259,-56.688,-179.895,7.621,149.408
C02440=1104.456,68.509,-56.706,-179.894,7.625,149.408
C02441=1104.451,68.758,-56.724,-179.893,7.628,149.409
C02442=1104.446,69.007,-56.742,-179.892,7.632,149.410
C02443=1104.441,69.257,-56.759,-179.890,7.636,149.410
C02444=1104.436,69.506,-56.777,-179.889,7.640,149.410
C02445=1104.431,69.755,-56.795,-179.888,7.644,149.411
C02446=1104.426,70.004,-56.813,-179.886,7.648,149.411
C02447=1104.422,70.254,-56.831,-179.885,7.652,149.412
C02448=1104.417,70.503,-56.849,-179.884,7.656,149.413
C02449=1104.412,70.753,-56.867,-179.882,7.660,149.413
C02450=1104.407,71.002,-56.885,-179.881,7.664,149.414
C02451=1104.402,71.251,-56.903,-179.880,7.668,149.414
C02452=1104.397,71.500,-56.921,-179.878,7.672,149.415
C02453=1104.393,71.750,-56.940,-179.877,7.676,149.415
C02454=1104.388,71.999,-56.958,-179.875,7.680,149.416
C02455=1104.383,72.248,-56.976,-179.874,7.683,149.416
C02456=1104.378,72.497,-56.994,-179.873,7.687,149.417
C02457=1104.373,72.746,-57.012,-179.872,7.691,149.417
C02458=1104.368,72.996,-57.031,-179.870,7.695,149.418
C02459=1104.363,73.245,-57.049,-179.869,7.699,149.418
C02460=1104.359,73.495,-57.067,-179.867,7.703,149.419
C02461=1104.354,73.744,-57.085,-179.866,7.707,149.419
C02462=1104.349,73.993,-57.103,-179.864,7.711,149.420
C02463=1104.344,74.243,-57.122,-179.864,7.715,149.420
C02464=1104.340,74.492,-57.140,-179.862,7.718,149.421
C02465=1104.335,74.740,-57.158,-179.861,7.722,149.421
C02466=1104.329,74.990,-57.177,-179.860,7.727,149.422
C02467=1104.325,75.240,-57.195,-179.858,7.731,149.422
C02468=1104.320,75.489,-57.213,-179.856,7.734,149.423
C02469=1104.315,75.738,-57.231,-179.855,7.739,149.423
C02470=1104.311,75.987,-57.250,-179.854,7.743,149.424
C02471=1104.305,76.237,-57.269,-179.852,7.747,149.424
C02472=1104.301,76.486,-57.287,-179.851,7.750,149.425
C02473=1104.296,76.735,-57.305,-179.849,7.755,149.425
C02474=1104.291,76.984,-57.323,-179.848,7.758,149.426
C02475=1104.287,77.198,-57.339,-179.848,7.761,149.426
C02476=1104.283,77.411,-57.355,-179.847,7.764,149.426
C02477=1104.278,77.625,-57.371,-179.846,7.768,149.427
C02478=1104.275,77.839,-57.387,-179.845,7.771,149.428
C02479=1104.270,78.052,-57.403,-179.844,7.774,149.428
C02480=1104.266,78.265,-57.418,-179.843,7.777,149.428
C02481=1104.263,78.479,-57.434,-179.842,7.780,149.429
C02482=1104.258,78.693,-57.450,-179.842,7.783,149.430
C02483=1104.253,78.942,-57.468,-179.840,7.787,149.430
C02484=1104.248,79.192,-57.487,-179.840,7.791,149.431
C02485=1104.244,79.441,-57.505,-179.838,7.795,149.431
C02486=1104.239,79.690,-57.523,-179.838,7.798,149.432
C02487=1104.234,79.939,-57.543,-179.836,7.802,149.432
C02488=1104.229,80.189,-57.561,-179.835,7.806,149.433
C02489=1104.224,80.438,-57.579,-179.834,7.810,149.433
C02490=1104.219,80.687,-57.599,-179.833,7.813,149.434
C02491=1104.215,80.937,-57.617,-179.832,7.817,149.435
C02492=1104.210,81.185,-57.635,-179.831,7.820,149.435
C02493=1104.205,81.435,-57.654,-179.830,7.825,149.436
C02494=1104.200,81.684,-57.672,-179.829,7.828,149.436
C02495=1104.196,81.934,-57.691,-179.828,7.832,149.437
C02496=1104.190,82.183,-57.710,-179.827,7.835,149.437
C02497=1104.186,82.432,-57.729,-179.826,7.840,149.438
C02498=1104.181,82.682,-57.747,-179.825,7.843,149.438
C02499=1104.176,82.930,-57.766,-179.824,7.847,149.439
C02500=1104.171,83.180,-57.784,-179.822,7.851,149.439
C02501=1104.167,83.429,-57.803,-179.822,7.854,149.440
C02502=1104.161,83.678,-57.822,-179.820,7.858,149.440
C02503=1104.157,83.928,-57.841,-179.820,7.862,149.441
C02504=1104.152,84.177,-57.859,-179.818,7.866,149.441
C02505=1104.147,84.426,-57.878,-179.818,7.869,149.442
C02506=1104.143,84.676,-57.896,-179.816,7.873,149.443
C02507=1104.138,84.924,-57.916,-179.815,7.877,149.443
C02508=1104.134,85.174,-57.935,-179.814,7.880,149.444
C02509=1104.128,85.423,-57.953,-179.812,7.884,149.444
C02510=1104.124,85.672,-57.972,-179.812,7.888,149.445
C02511=1104.118,85.922,-57.991,-179.810,7.892,149.445
C02512=1104.114,86.170,-58.010,-179.809,7.896,149.446
C02513=1104.109,86.420,-58.029,-179.808,7.899,149.446
C02514=1104.104,86.669,-58.047,-179.807,7.903,149.447
C02515=1104.099,86.919,-58.067,-179.806,7.906,149.447
C02516=1104.095,87.167,-58.086,-179.805,7.911,149.448
C02517=1104.090,87.417,-58.104,-179.803,7.915,149.448
C02518=1104.085,87.666,-58.123,-179.802,7.918,149.449
C02519=1104.081,87.915,-58.142,-179.801,7.922,149.450
C02520=1104.075,88.165,-58.161,-179.800,7.926,149.450
C02521=1104.071,88.414,-58.181,-179.799,7.929,149.450
C02522=1104.066,88.663,-58.199,-179.797,7.933,149.451
C02523=1104.060,88.912,-58.218,-179.796,7.937,149.451
C02524=1104.056,89.162,-58.237,-179.795,7.941,149.452
C02525=1104.051,89.411,-58.256,-179.794,7.944,149.453
C02526=1104.047,89.660,-58.275,-179.793,7.948,149.453
C02527=1104.041,89.909,-58.294,-179.792,7.952,149.454
C02528=1104.037,90.159,-58.313,-179.790,7.956,149.454
C02529=1104.033,90.408,-58.333,-179.789,7.959,149.455
C02530=1104.028,90.657,-58.351,-179.788,7.963,149.455
C02531=1104.023,90.871,-58.368,-179.787,7.966,149.456
C02532=1104.019,91.084,-58.384,-179.786,7.969,149.456
C02533=1104.015,91.298,-58.401,-179.784,7.973,149.456
C02534=1104.011,91.511,-58.417,-179.783,7.976,149.457
C02535=1104.008,91.725,-58.433,-179.782,7.979,149.457
C02536=1104.003,91.938,-58.450,-179.781,7.982,149.458
C02537=1103.999,92.152,-58.466,-179.780,7.985,149.458
C02538=1103.995,92.365,-58.483,-179.779,7.988,149.458
C02539=1103.990,92.614,-58.502,-179.778,7.992,149.459
C02540=1103.985,92.863,-58.521,-179.776,7.997,149.460
C02541=1103.980,93.113,-58.540,-179.775,8.000,149.460
C02542=1103.975,93.362,-58.559,-179.774,8.004,149.460
C02543=1103.971,93.611,-58.578,-179.772,8.007,149.461
C02544=1103.966,93.860,-58.598,-179.771,8.012,149.461
C02545=1103.961,94.110,-58.617,-179.770,8.015,149.462
C02546=1103.957,94.359,-58.636,-179.769,8.019,149.462
C02547=1103.952,94.608,-58.656,-179.767,8.023,149.463
C02548=1103.947,94.857,-58.675,-179.766,8.026,149.463
C02549=1103.942,95.106,-58.694,-179.765,8.030,149.464
C02550=1103.937,95.355,-58.714,-179.763,8.034,149.464
C02551=1103.933,95.605,-58.733,-179.762,8.038,149.465
C02552=1103.928,95.854,-58.752,-179.761,8.041,149.465
C02553=1103.923,96.103,-58.772,-179.759,8.045,149.466
C02554=1103.918,96.352,-58.791,-179.757,8.049,149.466
C02555=1103.913,96.602,-58.811,-179.756,8.053,149.466
C02556=1103.909,96.851,-58.830,-179.755,8.056,149.467
C02557=1103.904,97.100,-58.849,-179.753,8.060,149.467
C02558=1103.899,97.349,-58.869,-179.752,8.064,149.468
C02559=1103.894,97.599,-58.888,-179.751,8.068,149.468
C02560=1103.889,97.848,-58.908,-179.750,8.071,149.469
C02561=1103.885,98.096,-58.927,-179.748,8.075,149.469
C02562=1103.881,98.346,-58.947,-179.746,8.079,149.470
C02563=1103.875,98.595,-58.966,-179.745,8.082,149.470
C02564=1103.871,98.844,-58.986,-179.744,8.086,149.471
C02565=1103.866,99.094,-59.006,-179.742,8.089,149.471
C02566=1103.861,99.342,-59.024,-179.741,8.093,149.472
C02567=1103.857,99.592,-59.044,-179.739,8.097,149.472
C02568=1103.852,99.841,-59.064,-179.738,8.100,149.472
C02569=1103.847,100.090,-59.084,-179.736,8.104,149.473
C02570=1103.842,100.339,-59.103,-179.735,8.108,149.473
C02571=1103.837,100.589,-59.123,-179.733,8.112,149.474
C02572=1103.833,100.838,-59.142,-179.731,8.115,149.474
C02573=1103.828,101.087,-59.162,-179.730,8.119,149.474
C02574=1103.823,101.336,-59.182,-179.729,8.122,149.475
C02575=1103.819,101.586,-59.201,-179.727,8.126,149.475
C02576=1103.813,101.835,-59.221,-179.725,8.130,149.476
C02577=1103.809,102.083,-59.241,-179.724,8.133,149.476
C02578=1103.804,102.333,-59.261,-179.723,8.137,149.477
C02579=1103.799,102.582,-59.280,-179.721,8.141,149.477
C02580=1103.794,102.831,-59.300,-179.719,8.145,149.477
C02581=1103.790,103.080,-59.320,-179.717,8.148,149.478
C02582=1103.785,103.330,-59.340,-179.717,8.152,149.478
C02583=1103.780,103.578,-59.360,-179.715,8.155,149.479
C02584=1103.775,103.828,-59.379,-179.713,8.159,149.479
C02585=1103.771,104.077,-59.398,-179.711,8.163,149.479
C02586=1103.767,104.326,-59.419,-179.710,8.167,149.480
C02587=1103.761,104.580,-59.438,-179.709,8.170,149.480
C02588=1103.757,104.835,-59.459,-179.707,8.174,149.480
C02589=1103.752,105.089,-59.479,-179.705,8.177,149.481
C02590=1103.747,105.342,-59.500,-179.703,8.181,149.481
C02591=1103.742,105.592,-59.519,-179.702,8.185,149.482
C02592=1103.737,105.841,-59.540,-179.700,8.189,149.482
C02593=1103.733,106.090,-59.559,-179.698,8.192,149.482
C02594=1103.728,106.339,-59.580,-179.697,8.195,149.483
C02595=1103.723,106.588,-59.599,-179.695,8.199,149.483
C02596=1103.718,106.837,-59.619,-179.693,8.203,149.483
C02597=1103.714,107.087,-59.639,-179.691,8.206,149.484
C02598=1103.709,107.336,-59.659,-179.690,8.210,149.484
C02599=1103.704,107.585,-59.679,-179.689,8.213,149.484
C02600=1103.700,107.834,-59.699,-179.687,8.217,149.485
C02601=1103.695,108.083,-59.719,-179.685,8.221,149.485
C02602=1103.690,108.332,-59.739,-179.683,8.224,149.485
C02603=1103.685,108.582,-59.759,-179.681,8.228,149.486
C02604=1103.680,108.831,-59.780,-179.680,8.231,149.486
C02605=1103.676,109.080,-59.799,-179.678,8.235,149.486
C02606=1103.671,109.329,-59.820,-179.676,8.238,149.487
C02607=1103.667,109.578,-59.840,-179.675,8.242,149.487
C02608=1103.661,109.827,-59.859,-179.673,8.246,149.487
C02609=1103.657,110.076,-59.880,-179.671,8.249,149.488
C02610=1103.652,110.325,-59.901,-179.670,8.252,149.488
C02611=1103.647,110.575,-59.920,-179.668,8.256,149.488
C02612=1103.643,110.824,-59.941,-179.666,8.260,149.489
C02613=1103.638,111.073,-59.961,-179.664,8.263,149.489
C02614=1103.633,111.322,-59.981,-179.662,8.267,149.489
C02615=1103.629,111.571,-60.001,-179.661,8.270,149.490
C02616=1103.624,111.821,-60.022,-179.659,8.273,149.490
C02617=1103.619,112.070,-60.042,-179.657,8.277,149.490
C02618=1103.614,112.318,-60.062,-179.656,8.280,149.490
C02619=1103.610,112.567,-60.082,-179.654,8.283,149.491
C02620=1103.604,112.817,-60.103,-179.652,8.287,149.491
C02621=1103.600,113.066,-60.123,-179.651,8.290,149.491
C02622=1103.595,113.315,-60.143,-179.649,8.294,149.492
C02623=1103.366,103.256,-59.385,-179.713,8.153,149.477
C02624=1103.371,103.007,-59.364,-179.715,8.149,149.477
C02625=1103.375,102.757,-59.345,-179.717,8.145,149.477
C02626=1103.380,102.508,-59.325,-179.717,8.142,149.476
C02627=1103.385,102.260,-59.305,-179.720,8.138,149.476
C02628=1103.390,102.010,-59.285,-179.721,8.135,149.475
C02629=1103.395,101.760,-59.266,-179.723,8.131,149.475
C02630=1103.399,101.511,-59.246,-179.724,8.128,149.475
C02631=1103.404,101.263,-59.227,-179.725,8.124,149.474
C02632=1103.408,101.013,-59.207,-179.727,8.120,149.474
C02633=1103.413,100.764,-59.187,-179.729,8.116,149.473
C02634=1103.418,100.514,-59.168,-179.730,8.112,149.473
C02635=1103.423,100.266,-59.148,-179.731,8.109,149.472
C02636=1103.428,100.016,-59.128,-179.733,8.105,149.472
C02637=1103.432,99.767,-59.108,-179.734,8.101,149.472
C02638=1103.438,99.518,-59.089,-179.736,8.098,149.471
C02639=1103.442,99.269,-59.070,-179.737,8.095,149.471
C02640=1103.446,99.020,-59.050,-179.739,8.091,149.470
C02641=1103.452,98.771,-59.030,-179.741,8.087,149.470
C02642=1103.456,98.521,-59.011,-179.742,8.082,149.469
C02643=1103.461,98.272,-58.991,-179.743,8.079,149.469
C02644=1103.466,98.023,-58.972,-179.744,8.075,149.468
C02645=1103.470,97.774,-58.953,-179.746,8.072,149.468
C02646=1103.475,97.524,-58.933,-179.747,8.068,149.468
C02647=1103.481,97.275,-58.914,-179.748,8.065,149.467
C02648=1103.485,97.026,-58.893,-179.750,8.061,149.467
C02649=1103.489,96.777,-58.874,-179.752,8.057,149.466
C02650=1103.494,96.528,-58.855,-179.753,8.053,149.466
C02651=1103.499,96.279,-58.835,-179.754,8.050,149.465
C02652=1103.504,96.029,-58.816,-179.756,8.046,149.465
C02653=1103.508,95.780,-58.797,-179.757,8.042,149.465
C02654=1103.513,95.531,-58.777,-179.758,8.039,149.464
C02655=1103.518,95.282,-58.758,-179.760,8.035,149.463
C02656=1103.523,95.032,-58.738,-179.761,8.031,149.463
C02657=1103.527,94.783,-58.719,-179.763,8.027,149.463
C02658=1103.533,94.534,-58.700,-179.764,8.024,149.462
C02659=1103.537,94.285,-58.680,-179.765,8.020,149.462
C02660=1103.542,94.036,-58.662,-179.766,8.016,149.461
C02661=1103.547,93.787,-58.642,-179.767,8.013,149.461
C02662=1103.551,93.537,-58.622,-179.769,8.009,149.460
C02663=1103.556,93.289,-58.604,-179.771,8.005,149.460
C02664=1103.561,93.038,-58.585,-179.772,8.001,149.459
C02665=1103.566,92.789,-58.566,-179.773,7.997,149.459
C02666=1103.570,92.540,-58.546,-179.774,7.993,149.458
C02667=1103.576,92.291,-58.527,-179.776,7.990,149.458
C02668=1103.583,91.884,-58.495,-179.778,7.983,149.457
C02669=1103.591,91.476,-58.464,-179.780,7.977,149.456
C02670=1103.599,91.070,-58.433,-179.782,7.971,149.455
C02671=1103.607,90.662,-58.402,-179.784,7.965,149.455
C02672=1103.611,90.414,-58.383,-179.785,7.962,149.454
C02673=1103.616,90.164,-58.363,-179.786,7.958,149.453
C02674=1103.622,89.915,-58.345,-179.788,7.954,149.453
C02675=1103.626,89.665,-58.326,-179.788,7.950,149.452
C02676=1103.631,89.416,-58.306,-179.790,7.946,149.452
C02677=1103.635,89.167,-58.287,-179.792,7.943,149.451
C02678=1103.640,88.918,-58.268,-179.792,7.939,149.451
C02679=1103.645,88.668,-58.250,-179.794,7.935,149.450
C02680=1103.650,88.420,-58.230,-179.795,7.931,149.450
C02681=1103.654,88.170,-58.211,-179.796,7.928,149.449
C02682=1103.660,87.921,-58.193,-179.797,7.924,149.449
C02683=1103.664,87.672,-58.174,-179.798,7.921,149.448
C02684=1103.669,87.423,-58.154,-179.799,7.917,149.448
C02685=1103.673,87.173,-58.136,-179.801,7.913,149.447
C02686=1103.679,86.924,-58.117,-179.802,7.909,149.447
C02687=1103.683,86.675,-58.098,-179.803,7.905,149.446
C02688=1103.688,86.425,-58.079,-179.804,7.901,149.446
C02689=1103.692,86.176,-58.060,-179.805,7.898,149.445
C02690=1103.698,85.927,-58.041,-179.807,7.894,149.445
C02691=1103.703,85.678,-58.023,-179.807,7.890,149.444
C02692=1103.707,85.428,-58.003,-179.809,7.887,149.444
C02693=1103.712,85.180,-57.984,-179.810,7.882,149.443
C02694=1103.717,84.930,-57.965,-179.811,7.879,149.443
C02695=1103.722,84.681,-57.947,-179.812,7.875,149.442
C02696=1103.727,84.431,-57.928,-179.813,7.872,149.442
C02697=1103.731,84.182,-57.909,-179.814,7.868,149.441
C02698=1103.736,83.933,-57.891,-179.815,7.864,149.440
C02699=1103.741,83.684,-57.872,-179.816,7.860,149.440
C02700=1103.746,83.435,-57.853,-179.818,7.856,149.439
C02701=1103.751,83.185,-57.834,-179.818,7.853,149.439
C02702=1103.755,82.936,-57.815,-179.820,7.849,149.438
C02703=1103.760,82.687,-57.797,-179.821,7.845,149.438
C02704=1103.765,82.438,-57.778,-179.822,7.841,149.437
C02705=1103.770,82.188,-57.760,-179.823,7.838,149.437
C02706=1103.774,81.939,-57.741,-179.824,7.834,149.436
C02707=1103.780,81.690,-57.722,-179.825,7.831,149.435
C02708=1103.784,81.440,-57.704,-179.826,7.827,149.435
C02709=1103.788,81.191,-57.685,-179.827,7.823,149.434
C02710=1103.794,80.942,-57.666,-179.828,7.819,149.434
C02711=1103.799,80.693,-57.648,-179.829,7.816,149.433
C02712=1103.803,80.443,-57.629,-179.831,7.812,149.433
C02713=1103.808,80.194,-57.610,-179.832,7.808,149.432
C02714=1103.813,79.945,-57.592,-179.833,7.805,149.432
C02715=1103.818,79.695,-57.574,-179.834,7.800,149.431
C02716=1103.823,79.446,-57.554,-179.834,7.797,149.430
C02717=1103.828,79.197,-57.536,-179.836,7.793,149.430
C02718=1103.832,78.948,-57.517,-179.836,7.789,149.429
C02719=1103.837,78.699,-57.499,-179.837,7.786,149.429
C02720=1103.841,78.485,-57.484,-179.838,7.783,149.428
C02721=1103.845,78.271,-57.468,-179.839,7.780,149.428
C02722=1103.849,78.058,-57.452,-179.840,7.777,149.427
C02723=1103.854,77.845,-57.436,-179.841,7.773,149.427
C02724=1103.858,77.630,-57.420,-179.842,7.770,149.427
C02725=1103.862,77.417,-57.404,-179.843,7.767,149.426
C02726=1103.866,77.204,-57.388,-179.843,7.764,149.425
C02727=1103.870,76.990,-57.372,-179.844,7.761,149.425
C02728=1103.875,76.740,-57.354,-179.846,7.757,149.425
C02729=1103.880,76.492,-57.336,-179.847,7.753,149.424
C02730=1103.885,76.243,-57.318,-179.848,7.749,149.423
C02731=1103.890,75.993,-57.299,-179.850,7.745,149.423
C02732=1103.894,75.744,-57.280,-179.851,7.741,149.423
C02733=1103.899,75.495,-57.262,-179.853,7.736,149.422
C02734=1103.904,75.245,-57.244,-179.854,7.733,149.422
C02735=1103.909,74.996,-57.226,-179.855,7.729,149.421
C02736=1103.913,74.747,-57.208,-179.857,7.726,149.421
C02737=1103.919,74.498,-57.189,-179.858,7.721,149.420
C02738=1103.923,74.248,-57.170,-179.859,7.717,149.420
C02739=1103.928,73.999,-57.152,-179.861,7.713,149.419
C02740=1103.933,73.749,-57.134,-179.862,7.709,149.418
C02741=1103.938,73.500,-57.116,-179.864,7.705,149.418
C02742=1103.943,73.251,-57.098,-179.865,7.701,149.418
C02743=1103.947,73.001,-57.080,-179.866,7.697,149.417
C02744=1103.952,72.753,-57.061,-179.867,7.694,149.416
C02745=1103.957,72.503,-57.043,-179.869,7.690,149.416
C02746=1103.962,72.254,-57.025,-179.870,7.686,149.415
C02747=1103.967,72.005,-57.007,-179.872,7.682,149.415
C02748=1103.971,71.755,-56.988,-179.873,7.678,149.415
C02749=1103.976,71.506,-56.970,-179.874,7.674,149.414
C02750=1103.981,71.257,-56.952,-179.876,7.670,149.413
C02751=1103.986,71.007,-56.934,-179.877,7.666,149.413
C02752=1103.991,70.758,-56.916,-179.878,7.662,149.412
C02753=1103.995,70.508,-56.898,-179.879,7.658,149.412
C02754=1104.000,70.259,-56.880,-179.881,7.655,149.411
C02755=1104.005,70.010,-56.862,-179.882,7.650,149.411
C02756=1104.010,69.761,-56.844,-179.884,7.646,149.410
C02757=1104.015,69.512,-56.826,-179.885,7.643,149.410
C02758=1104.020,69.263,-56.808,-179.886,7.638,149.409
C02759=1104.025,69.013,-56.790,-179.887,7.635,149.409
C02760=1104.029,68.763,-56.772,-179.888,7.631,149.408
C02761=1104.034,68.514,-56.754,-179.890,7.627,149.408
C02762=1104.039,68.265,-56.736,-179.892,7.623,149.407
C02763=1104.044,68.016,-56.718,-179.893,7.619,149.407
C02764=1104.049,67.766,-56.701,-179.894,7.615,149.406
C02765=1104.054,67.517,-56.683,-179.895,7.612,149.406
C02766=1104.059,67.268,-56.665,-179.896,7.607,149.405
C02767=1104.064,67.019,-56.647,-179.898,7.604,149.405
C02768=1104.069,66.769,-56.629,-179.899,7.599,149.404
C02769=1104.073,66.520,-56.610,-179.901,7.595,149.404
C02770=1104.078,66.270,-56.592,-179.902,7.591,149.403
C02771=1104.083,66.021,-56.575,-179.903,7.588,149.403
C02772=1104.088,65.771,-56.557,-179.904,7.584,149.402
C02773=1104.092,65.523,-56.540,-179.905,7.580,149.401
C02774=1104.097,65.273,-56.522,-179.907,7.576,149.401
C02775=1104.102,65.024,-56.504,-179.908,7.572,149.401
C02776=1104.107,64.810,-56.489,-179.909,7.568,149.400
C02777=1104.111,64.597,-56.474,-179.910,7.565,149.400
C02778=1104.115,64.382,-56.458,-179.911,7.561,149.399
C02779=1104.118,64.169,-56.443,-179.912,7.558,149.399
C02780=1104.123,63.955,-56.428,-179.913,7.555,149.398
C02781=1104.127,63.742,-56.412,-179.914,7.552,149.398
C02782=1104.131,63.528,-56.398,-179.916,7.548,149.397
C02783=1104.136,63.315,-56.382,-179.917,7.545,149.397
C02784=1104.140,63.066,-56.365,-179.918,7.541,149.396
C02785=1104.145,62.816,-56.348,-179.919,7.538,149.396
C02786=1104.150,62.567,-56.330,-179.920,7.533,149.395
C02787=1104.155,62.318,-56.312,-179.921,7.529,149.395
C02788=1104.160,62.068,-56.294,-179.923,7.525,149.394
C02789=1104.165,61.819,-56.276,-179.924,7.521,149.394
C02790=1104.169,61.570,-56.259,-179.925,7.518,149.393
C02791=1104.175,61.320,-56.242,-179.926,7.514,149.393
C02792=1104.180,61.071,-56.224,-179.928,7.510,149.392
C02793=1104.185,60.821,-56.206,-179.929,7.506,149.391
C02794=1104.189,60.572,-56.189,-179.930,7.502,149.391
C02795=1104.194,60.323,-56.171,-179.931,7.498,149.390
C02796=1104.199,60.073,-56.154,-179.932,7.494,149.390
C02797=1104.204,59.824,-56.136,-179.934,7.490,149.389
C02798=1104.208,59.575,-56.119,-179.935,7.486,149.389
C02799=1104.213,59.326,-56.101,-179.936,7.482,149.388
C02800=1104.219,59.076,-56.084,-179.937,7.478,149.388
C02801=1104.223,58.827,-56.067,-179.938,7.474,149.387
C02802=1104.228,58.577,-56.049,-179.939,7.470,149.386
C02803=1104.233,58.328,-56.031,-179.941,7.466,149.386
C02804=1104.238,58.078,-56.014,-179.941,7.463,149.385
C02805=1104.242,57.829,-55.997,-179.943,7.459,149.385
C02806=1104.247,57.579,-55.979,-179.944,7.454,149.384
C02807=1104.252,57.330,-55.961,-179.946,7.451,149.384
C02808=1104.257,57.081,-55.945,-179.947,7.446,149.383
C02809=1104.262,56.832,-55.927,-179.948,7.443,149.383
C02810=1104.268,56.583,-55.910,-179.949,7.439,149.382
C02811=1104.272,56.334,-55.893,-179.950,7.435,149.381
C02812=1104.277,56.084,-55.875,-179.951,7.431,149.381
C02813=1104.281,55.834,-55.859,-179.952,7.427,149.380
C02814=1104.286,55.585,-55.841,-179.953,7.423,149.380
C02815=1104.292,55.335,-55.823,-179.954,7.419,149.379
C02816=1104.296,55.086,-55.807,-179.956,7.415,149.379
C02817=1104.301,54.837,-55.789,-179.957,7.412,149.378
C02818=1104.306,54.588,-55.772,-179.958,7.407,149.377
C02819=1104.311,54.338,-55.755,-179.959,7.403,149.377
C02820=1104.316,54.089,-55.737,-179.960,7.399,149.376
C02821=1104.321,53.840,-55.720,-179.961,7.396,149.376
C02822=1104.326,53.590,-55.703,-179.962,7.392,149.375
C02823=1104.330,53.341,-55.686,-179.963,7.387,149.375
C02824=1104.336,53.092,-55.669,-179.965,7.383,149.374
C02825=1104.340,52.842,-55.652,-179.965,7.380,149.374
C02826=1104.345,52.593,-55.634,-179.966,7.376,149.373
C02827=1104.351,52.343,-55.617,-179.968,7.372,149.372
C02828=1104.355,52.094,-55.600,-179.969,7.367,149.372
C02829=1104.360,51.844,-55.583,-179.970,7.364,149.371
C02830=1104.365,51.596,-55.566,-179.971,7.360,149.371
C02831=1104.370,51.346,-55.549,-179.972,7.356,149.370
C02832=1104.374,51.132,-55.534,-179.973,7.353,149.370
C02833=1104.378,50.919,-55.520,-179.974,7.349,149.369
C02834=1104.382,50.705,-55.506,-179.975,7.345,149.369
C02835=1104.387,50.491,-55.490,-179.976,7.342,149.368
C02836=1104.391,50.277,-55.476,-179.977,7.338,149.367
C02837=1104.395,50.064,-55.462,-179.978,7.335,149.367
C02838=1104.399,49.850,-55.447,-179.978,7.332,149.367
C02839=1104.404,49.636,-55.432,-179.980,7.328,149.366
C02840=1104.408,49.386,-55.416,-179.980,7.325,149.365
C02841=1104.414,49.137,-55.399,-179.982,7.321,149.365
C02842=1104.418,48.888,-55.382,-179.983,7.316,149.364
C02843=1104.423,48.638,-55.365,-179.983,7.313,149.364
C02844=1104.428,48.389,-55.347,-179.985,7.309,149.363
C02845=1104.433,48.140,-55.331,-179.986,7.305,149.362
C02846=1104.438,47.891,-55.314,-179.987,7.300,149.362
C02847=1104.443,47.641,-55.297,-179.987,7.297,149.361
C02848=1104.447,47.392,-55.280,-179.989,7.293,149.361
C02849=1104.453,47.142,-55.264,-179.990,7.288,149.360
C02850=1104.457,46.893,-55.247,-179.991,7.284,149.359
C02851=1104.462,46.644,-55.230,-179.991,7.281,149.359
C02852=1104.467,46.394,-55.213,-179.993,7.277,149.358
C02853=1104.472,46.145,-55.197,-179.994,7.272,149.358
C02854=1104.477,45.895,-55.179,-179.995,7.269,149.357
C02855=1104.482,45.646,-55.163,-179.996,7.265,149.356
C02856=1104.487,45.397,-55.146,-179.997,7.260,149.356
C02857=1104.492,45.147,-55.129,-179.998,7.256,149.355
C02858=1104.497,44.898,-55.112,-179.999,7.253,149.355
C02859=1104.501,44.648,-55.096,-180.000,7.249,149.354
C02860=1104.506,44.399,-55.079,179.999,7.244,149.353
C02861=1104.511,44.150,-55.062,179.999,7.241,149.353
C02862=1104.516,43.900,-55.046,179.998,7.237,149.352
C02863=1104.521,43.651,-55.029,179.996,7.233,149.352
C02864=1104.526,43.401,-55.012,179.995,7.228,149.351
C02865=1104.531,43.152,-54.995,179.995,7.225,149.350
C02866=1104.536,42.903,-54.980,179.993,7.220,149.350
C02867=1104.540,42.653,-54.963,179.992,7.216,149.349
C02868=1104.546,42.403,-54.946,179.992,7.213,149.348
C02869=1104.551,42.155,-54.929,179.991,7.208,149.348
C02870=1104.555,41.905,-54.913,179.990,7.204,149.347
C02871=1104.560,41.656,-54.896,179.989,7.200,149.346
C02872=1104.566,41.406,-54.879,179.988,7.197,149.346
C02873=1104.570,41.156,-54.863,179.987,7.192,149.345
C02874=1104.575,40.908,-54.847,179.986,7.188,149.345
C02875=1104.580,40.658,-54.830,179.985,7.185,149.344
C02876=1104.585,40.408,-54.813,179.984,7.180,149.343
C02877=1104.590,40.160,-54.797,179.983,7.176,149.343
C02878=1104.595,39.909,-54.781,179.983,7.172,149.342
C02879=1104.600,39.661,-54.764,179.981,7.168,149.341
C02880=1104.605,39.411,-54.748,179.980,7.164,149.341
C02881=1104.609,39.162,-54.731,179.979,7.159,149.340
C02882=1104.615,38.912,-54.715,179.979,7.156,149.339
C02883=1104.620,38.662,-54.698,179.978,7.152,149.339
C02884=1104.625,38.414,-54.682,179.977,7.147,149.338
C02885=1104.629,38.164,-54.666,179.976,7.144,149.337
C02886=1104.634,37.914,-54.649,179.975,7.140,149.337
C02887=1104.639,37.665,-54.633,179.974,7.135,149.336
C02888=1104.643,37.451,-54.619,179.974,7.132,149.335
C02889=1104.647,37.237,-54.605,179.973,7.129,149.335
C02890=1104.652,37.024,-54.592,179.972,7.125,149.334
C02891=1104.656,36.810,-54.577,179.971,7.122,149.334
C02892=1104.660,36.596,-54.563,179.970,7.118,149.333
C02893=1104.664,36.382,-54.549,179.970,7.114,149.332
C02894=1104.668,36.168,-54.535,179.969,7.111,149.332
C02895=1104.673,35.955,-54.521,179.969,7.107,149.331
C02896=1104.678,35.705,-54.505,179.967,7.103,149.331
C02897=1104.683,35.456,-54.489,179.967,7.100,149.330
C02898=1104.688,35.206,-54.472,179.966,7.095,149.329
C02899=1104.693,34.957,-54.456,179.965,7.091,149.329
C02900=1104.698,34.707,-54.439,179.964,7.087,149.328
C02901=1104.703,34.458,-54.423,179.963,7.083,149.327
C02902=1104.708,34.208,-54.407,179.962,7.079,149.327
C02903=1104.713,33.959,-54.391,179.962,7.074,149.326
C02904=1104.718,33.709,-54.375,179.961,7.071,149.325
C02905=1104.723,33.461,-54.359,179.960,7.066,149.325
C02906=1104.728,33.210,-54.343,179.959,7.062,149.324
C02907=1104.733,32.962,-54.326,179.959,7.059,149.323
C02908=1104.738,32.712,-54.310,179.958,7.054,149.323
C02909=1104.743,32.463,-54.294,179.957,7.050,149.322
C02910=1104.748,32.213,-54.278,179.957,7.046,149.321
C02911=1104.753,31.964,-54.262,179.956,7.042,149.320
C02912=1104.758,31.714,-54.246,179.954,7.037,149.320
C02913=1104.763,31.465,-54.230,179.954,7.034,149.319
C02914=1104.767,31.215,-54.214,179.953,7.030,149.318
C02915=1104.772,30.966,-54.197,179.952,7.025,149.318
C02916=1104.777,30.716,-54.181,179.952,7.021,149.317
C02917=1104.782,30.467,-54.166,179.951,7.017,149.316
C02918=1104.787,30.218,-54.150,179.950,7.013,149.316
C02919=1104.792,29.968,-54.134,179.949,7.008,149.315
C02920=1104.797,29.719,-54.118,179.949,7.005,149.314
C02921=1104.802,29.469,-54.102,179.948,7.000,149.313
C02922=1104.807,29.220,-54.086,179.947,6.996,149.313
C02923=1104.812,28.970,-54.070,179.947,6.992,149.312
C02924=1104.817,28.721,-54.054,179.946,6.988,149.311
C02925=1104.822,28.471,-54.039,179.945,6.983,149.311
C02926=1104.827,28.222,-54.022,179.944,6.980,149.310
C02927=1104.832,27.973,-54.006,179.944,6.975,149.309
C02928=1104.836,27.723,-53.991,179.943,6.971,149.308
C02929=1104.841,27.474,-53.975,179.942,6.967,149.308
C02930=1104.847,27.225,-53.959,179.942,6.963,149.307
C02931=1104.851,26.974,-53.943,179.940,6.958,149.306
C02932=1104.857,26.726,-53.927,179.940,6.955,149.306
C02933=1104.861,26.476,-53.911,179.939,6.950,149.305
C02934=1104.866,26.226,-53.896,179.938,6.946,149.304
C02935=1104.871,25.977,-53.880,179.938,6.942,149.303
C02936=1104.876,25.728,-53.864,179.937,6.938,149.302
C02937=1104.881,25.478,-53.848,179.936,6.933,149.302
C02938=1104.887,25.229,-53.832,179.936,6.929,149.301
C02939=1104.891,24.979,-53.816,179.935,6.925,149.300
C02940=1104.896,24.730,-53.801,179.935,6.920,149.299
C02941=1104.901,24.481,-53.785,179.934,6.916,149.299
C02942=1104.906,24.231,-53.769,179.933,6.913,149.298
C02943=1104.911,23.981,-53.754,179.933,6.908,149.297
C02944=1104.915,23.767,-53.740,179.932,6.904,149.296
C02945=1104.920,23.554,-53.727,179.932,6.901,149.296
C02946=1104.924,23.339,-53.713,179.931,6.897,149.295
C02947=1104.928,23.125,-53.700,179.930,6.893,149.295
C02948=1104.932,22.912,-53.687,179.930,6.890,149.294
C02949=1104.937,22.697,-53.673,179.929,6.886,149.293
C02950=1104.941,22.484,-53.660,179.929,6.882,149.293
C02951=1104.945,22.270,-53.646,179.929,6.879,149.292
C02952=1104.950,22.021,-53.630,179.928,6.875,149.291
C02953=1104.955,21.771,-53.615,179.927,6.870,149.290
C02954=1104.960,21.522,-53.600,179.927,6.866,149.290
C02955=1104.965,21.272,-53.584,179.926,6.862,149.289
C02956=1104.971,21.023,-53.568,179.925,6.857,149.288
C02957=1104.975,20.773,-53.553,179.925,6.853,149.287
C02958=1104.980,20.524,-53.537,179.924,6.849,149.287
C02959=1104.985,20.274,-53.522,179.923,6.844,149.286
C02960=1104.989,20.025,-53.506,179.923,6.841,149.285
C02961=1104.995,19.775,-53.491,179.922,6.836,149.284
C02962=1105.000,19.526,-53.475,179.922,6.832,149.283
C02963=1105.005,19.277,-53.460,179.921,6.828,149.283
C02964=1105.010,19.027,-53.444,179.921,6.823,149.282
C02965=1105.015,18.777,-53.429,179.920,6.819,149.281
C02966=1105.020,18.528,-53.414,179.920,6.815,149.280
C02967=1105.025,18.279,-53.398,179.919,6.810,149.279
C02968=1105.030,18.029,-53.382,179.918,6.806,149.279
C02969=1105.034,17.780,-53.367,179.918,6.801,149.278
C02970=1105.040,17.530,-53.352,179.918,6.797,149.277
C02971=1105.044,17.281,-53.337,179.917,6.793,149.276
C02972=1105.050,17.032,-53.321,179.916,6.788,149.275
C02973=1105.055,16.782,-53.305,179.916,6.785,149.274
C02974=1105.059,16.532,-53.290,179.915,6.780,149.274
C02975=1105.065,16.283,-53.275,179.915,6.776,149.273
C02976=1105.070,16.033,-53.260,179.915,6.772,149.272
C02977=1105.074,15.783,-53.244,179.914,6.767,149.271
C02978=1105.080,15.534,-53.229,179.913,6.763,149.270
C02979=1105.084,15.285,-53.214,179.913,6.759,149.270
C02980=1105.090,15.035,-53.198,179.912,6.754,149.269
C02981=1105.095,14.786,-53.183,179.912,6.749,149.268
C02982=1105.100,14.537,-53.168,179.911,6.745,149.267
C02983=1105.104,14.286,-53.153,179.911,6.741,149.266
C02984=1105.110,14.037,-53.137,179.910,6.736,149.265
C02985=1105.114,13.788,-53.122,179.910,6.732,149.264
C02986=1105.120,13.539,-53.107,179.910,6.728,149.264
C02987=1105.124,13.289,-53.092,179.909,6.723,149.263
C02988=1105.130,13.039,-53.077,179.908,6.719,149.262
C02989=1105.134,12.790,-53.062,179.908,6.715,149.261
C02990=1105.139,12.540,-53.046,179.908,6.710,149.260
C02991=1105.144,12.291,-53.031,179.907,6.705,149.259
C02992=1105.149,12.042,-53.015,179.907,6.701,149.258
C02993=1105.154,11.792,-53.001,179.907,6.697,149.258
C02994=1105.160,11.543,-52.985,179.906,6.692,149.257
C02995=1105.164,11.294,-52.970,179.905,6.688,149.256
C02996=1105.170,11.043,-52.956,179.905,6.684,149.255
C02997=1105.174,10.794,-52.940,179.905,6.679,149.254
C02998=1105.180,10.544,-52.925,179.904,6.674,149.253
C02999=1105.184,10.295,-52.910,179.904,6.671,149.253
C03000=1105.189,10.081,-52.898,179.903,6.666,149.252
C03001=1105.193,9.867,-52.884,179.903,6.662,149.251
C03002=1105.197,9.653,-52.872,179.903,6.659,149.250
C03003=1105.202,9.439,-52.858,179.903,6.655,149.249
C03004=1105.206,9.225,-52.845,179.902,6.651,149.249
C03005=1105.210,9.011,-52.833,179.902,6.647,149.248
C03006=1105.215,8.797,-52.820,179.902,6.643,149.247
C03007=1105.219,8.583,-52.807,179.901,6.640,149.247
C03008=1105.224,8.333,-52.792,179.901,6.635,149.246
C03009=1105.229,8.084,-52.777,179.900,6.630,149.245
C03010=1105.234,7.834,-52.762,179.899,6.625,149.244
C03011=1105.239,7.585,-52.747,179.899,6.621,149.243
C03012=1105.244,7.335,-52.733,179.898,6.616,149.242
C03013=1105.249,7.086,-52.718,179.897,6.612,149.241
C03014=1105.254,6.837,-52.702,179.897,6.607,149.241
C03015=1105.259,6.587,-52.688,179.896,6.602,149.240
C03016=1105.264,6.338,-52.673,179.895,6.598,149.239
C03017=1105.269,6.088,-52.658,179.895,6.593,149.238
C03018=1105.274,5.839,-52.643,179.894,6.589,149.237
C03019=1105.279,5.589,-52.629,179.894,6.584,149.236
C03020=1105.284,5.340,-52.613,179.893,6.580,149.236
C03021=1105.289,5.090,-52.599,179.892,6.575,149.235
C03022=1105.294,4.841,-52.584,179.892,6.570,149.234
C03023=1105.300,4.591,-52.569,179.891,6.565,149.233
C03024=1105.304,4.342,-52.554,179.890,6.561,149.232
C03025=1105.309,4.092,-52.540,179.889,6.556,149.231
C03026=1105.314,3.843,-52.525,179.889,6.552,149.231
C03027=1105.319,3.593,-52.510,179.888,6.547,149.230
C03028=1105.324,3.343,-52.495,179.887,6.543,149.229
C03029=1105.329,3.094,-52.480,179.887,6.538,149.228
C03030=1105.334,2.844,-52.466,179.886,6.533,149.227
C03031=1105.339,2.595,-52.451,179.885,6.529,149.227
C03032=1105.344,2.345,-52.436,179.885,6.524,149.226
C03033=1105.349,2.096,-52.422,179.884,6.519,149.225
C03034=1105.354,1.847,-52.407,179.884,6.515,149.224
C03035=1105.359,1.597,-52.393,179.883,6.510,149.223
C03036=1105.365,1.347,-52.378,179.882,6.506,149.222
C03037=1105.369,1.098,-52.363,179.882,6.501,149.221
C03038=1105.374,0.848,-52.349,179.881,6.497,149.221
C03039=1105.379,0.598,-52.334,179.881,6.493,149.220
C03040=1105.384,0.349,-52.319,179.880,6.488,149.219
C03041=1105.389,0.099,-52.305,179.880,6.483,149.218
C03042=1105.394,-0.151,-52.290,179.879,6.479,149.217
C03043=1105.400,-0.399,-52.276,179.878,6.474,149.216
C03044=1105.405,-0.649,-52.261,179.878,6.470,149.216
C03045=1105.410,-0.898,-52.247,179.877,6.465,149.215
C03046=1105.415,-1.148,-52.233,179.876,6.461,149.214
C03047=1105.419,-1.397,-52.218,179.876,6.456,149.213
C03048=1105.424,-1.647,-52.203,179.875,6.451,149.212
C03049=1105.430,-1.897,-52.189,179.874,6.447,149.212
C03050=1105.435,-2.147,-52.174,179.874,6.442,149.211
C03051=1105.440,-2.396,-52.160,179.873,6.437,149.210
C03052=1105.444,-2.645,-52.145,179.873,6.434,149.209
C03053=1105.450,-2.894,-52.131,179.872,6.429,149.208
C03054=1105.455,-3.144,-52.117,179.872,6.424,149.207
C03055=1105.460,-3.394,-52.103,179.871,6.420,149.207
C03056=1105.464,-3.608,-52.091,179.871,6.416,149.206
C03057=1105.468,-3.822,-52.078,179.870,6.412,149.205
C03058=1105.472,-4.036,-52.065,179.869,6.408,149.204
C03059=1105.478,-4.250,-52.053,179.869,6.405,149.204
C03060=1105.481,-4.465,-52.040,179.868,6.400,149.203
C03061=1105.486,-4.679,-52.028,179.868,6.396,149.202
C03062=1105.490,-4.892,-52.016,179.868,6.393,149.202
C03063=1105.495,-5.106,-52.004,179.867,6.389,149.201
C03064=1105.500,-5.356,-51.990,179.866,6.384,149.200
C03065=1105.505,-5.606,-51.976,179.865,6.380,149.199
C03066=1105.510,-5.856,-51.961,179.865,6.376,149.198
C03067=1105.514,-6.105,-51.946,179.865,6.371,149.198
C03068=1105.519,-6.354,-51.932,179.864,6.366,149.197
C03069=1105.525,-6.603,-51.918,179.863,6.362,149.196
C03070=1105.530,-6.853,-51.904,179.863,6.357,149.195
C03071=1105.535,-7.103,-51.890,179.862,6.352,149.194
C03072=1105.540,-7.352,-51.875,179.862,6.348,149.193
C03073=1105.545,-7.602,-51.861,179.861,6.343,149.193
C03074=1105.550,-7.851,-51.847,179.861,6.339,149.192
C03075=1105.555,-8.101,-51.833,179.860,6.335,149.191
C03076=1105.560,-8.351,-51.819,179.860,6.330,149.190
C03077=1105.565,-8.600,-51.804,179.859,6.326,149.189
C03078=1105.571,-8.849,-51.791,179.858,6.321,149.188
C03079=1105.576,-9.099,-51.776,179.858,6.316,149.187
C03080=1105.580,-9.348,-51.763,179.857,6.312,149.187
C03081=1105.585,-9.599,-51.749,179.857,6.308,149.186
C03082=1105.590,-9.848,-51.735,179.856,6.303,149.185
C03083=1105.596,-10.097,-51.721,179.856,6.299,149.184
C03084=1105.601,-10.347,-51.707,179.855,6.294,149.183
C03085=1105.605,-10.597,-51.692,179.854,6.290,149.183
C03086=1105.611,-10.846,-51.678,179.854,6.285,149.182
C03087=1105.616,-11.096,-51.664,179.853,6.280,149.181
C03088=1105.620,-11.345,-51.650,179.853,6.276,149.180
C03089=1105.625,-11.595,-51.636,179.853,6.271,149.179
C03090=1105.631,-11.844,-51.623,179.852,6.267,149.178
C03091=1105.636,-12.094,-51.609,179.851,6.262,149.177
C03092=1105.641,-12.344,-51.594,179.851,6.258,149.176
C03093=1105.646,-12.593,-51.580,179.850,6.253,149.176
C03094=1105.651,-12.842,-51.567,179.850,6.249,149.175
C03095=1105.656,-13.092,-51.553,179.850,6.244,149.174
C03096=1105.661,-13.342,-51.539,179.849,6.240,149.173
C03097=1105.666,-13.591,-51.525,179.849,6.235,149.172
C03098=1105.671,-13.841,-51.511,179.848,6.231,149.171
C03099=1105.676,-14.090,-51.497,179.848,6.226,149.170
C03100=1105.682,-14.340,-51.484,179.848,6.222,149.170
C03101=1105.686,-14.590,-51.470,179.847,6.217,149.169
C03102=1105.691,-14.839,-51.455,179.847,6.212,149.168
C03103=1105.696,-15.088,-51.442,179.846,6.208,149.167
C03104=1105.702,-15.338,-51.428,179.845,6.203,149.166
C03105=1105.706,-15.588,-51.414,179.845,6.199,149.165
C03106=1105.712,-15.837,-51.400,179.845,6.195,149.164
C03107=1105.717,-16.087,-51.387,179.844,6.190,149.163
C03108=1105.722,-16.337,-51.373,179.844,6.185,149.163
C03109=1105.727,-16.586,-51.359,179.843,6.181,149.162
C03110=1105.732,-16.836,-51.345,179.843,6.176,149.161
C03111=1105.737,-17.086,-51.332,179.842,6.171,149.160
C03112=1105.741,-17.300,-51.320,179.842,6.168,149.159
C03113=1105.745,-17.513,-51.308,179.842,6.164,149.158
C03114=1105.750,-17.728,-51.296,179.841,6.159,149.158
C03115=1105.755,-17.942,-51.284,179.841,6.156,149.157
C03116=1105.759,-18.156,-51.272,179.841,6.152,149.156
C03117=1105.763,-18.370,-51.262,179.840,6.148,149.155
C03118=1105.768,-18.584,-51.250,179.840,6.144,149.155
C03119=1105.772,-18.799,-51.237,179.840,6.140,149.154
C03120=1105.777,-19.048,-51.224,179.839,6.135,149.153
C03121=1105.782,-19.298,-51.210,179.839,6.131,149.152
C03122=1105.787,-19.547,-51.197,179.838,6.126,149.151
C03123=1105.792,-19.797,-51.183,179.838,6.122,149.150
C03124=1105.798,-20.046,-51.170,179.838,6.117,149.149
C03125=1105.802,-20.296,-51.156,179.837,6.113,149.148
C03126=1105.808,-20.546,-51.142,179.837,6.108,149.147
C03127=1105.813,-20.795,-51.129,179.836,6.103,149.147
C03128=1105.818,-21.045,-51.116,179.836,6.098,149.146
C03129=1105.823,-21.294,-51.102,179.836,6.094,149.145
C03130=1105.828,-21.544,-51.089,179.836,6.090,149.144
C03131=1105.833,-21.793,-51.075,179.835,6.085,149.143
C03132=1105.838,-22.043,-51.062,179.835,6.080,149.142
C03133=1105.844,-22.292,-51.048,179.834,6.075,149.141
C03134=1105.848,-22.543,-51.035,179.834,6.070,149.140
C03135=1105.854,-22.792,-51.021,179.834,6.066,149.139
C03136=1105.859,-23.042,-51.007,179.834,6.062,149.138
C03137=1105.863,-23.291,-50.994,179.833,6.057,149.137
C03138=1105.869,-23.541,-50.981,179.833,6.052,149.136
C03139=1105.873,-23.790,-50.967,179.832,6.048,149.135
C03140=1105.879,-24.040,-50.954,179.832,6.043,149.135
C03141=1105.884,-24.290,-50.941,179.832,6.038,149.133
C03142=1105.889,-24.539,-50.927,179.832,6.034,149.133
C03143=1105.894,-24.789,-50.914,179.831,6.029,149.132
C03144=1105.900,-25.039,-50.901,179.831,6.024,149.131
C03145=1105.904,-25.287,-50.887,179.831,6.020,149.130
C03146=1105.910,-25.538,-50.874,179.831,6.014,149.129
C03147=1105.914,-25.786,-50.861,179.830,6.010,149.128
C03148=1105.920,-26.037,-50.847,179.830,6.006,149.127
C03149=1105.925,-26.286,-50.834,179.830,6.001,149.126
C03150=1105.930,-26.536,-50.820,179.830,5.996,149.125
C03151=1105.935,-26.785,-50.807,179.830,5.992,149.124
C03152=1105.940,-27.035,-50.794,179.829,5.987,149.123
C03153=1105.945,-27.285,-50.781,179.829,5.983,149.122
C03154=1105.950,-27.534,-50.767,179.830,5.978,149.121
C03155=1105.955,-27.784,-50.754,179.829,5.974,149.120
C03156=1105.961,-28.034,-50.741,179.829,5.969,149.119
C03157=1105.965,-28.283,-50.728,179.829,5.965,149.118
C03158=1105.970,-28.533,-50.715,179.828,5.960,149.117
C03159=1105.976,-28.782,-50.701,179.828,5.955,149.116
C03160=1105.981,-29.032,-50.689,179.828,5.952,149.116
C03161=1105.986,-29.281,-50.675,179.827,5.947,149.115
C03162=1105.991,-29.531,-50.662,179.827,5.942,149.114
C03163=1105.996,-29.781,-50.649,179.827,5.938,149.113
C03164=1106.001,-30.030,-50.636,179.827,5.933,149.112
C03165=1106.006,-30.280,-50.623,179.826,5.929,149.111
C03166=1106.011,-30.529,-50.609,179.826,5.925,149.110
C03167=1106.017,-30.779,-50.596,179.826,5.920,149.109
C03168=1106.021,-30.993,-50.585,179.826,5.916,149.108
C03169=1106.025,-31.207,-50.574,179.826,5.913,149.108
C03170=1106.030,-31.421,-50.562,179.825,5.909,149.107
C03171=1106.034,-31.636,-50.551,179.826,5.905,149.106
C03172=1106.039,-31.850,-50.540,179.825,5.901,149.105
C03173=1106.043,-32.064,-50.529,179.824,5.897,149.105
C03174=1106.047,-32.279,-50.518,179.824,5.893,149.104
C03175=1106.051,-32.493,-50.507,179.824,5.890,149.103
C03176=1106.056,-32.743,-50.493,179.824,5.885,149.102
C03177=1106.062,-32.992,-50.481,179.824,5.881,149.101
C03178=1106.067,-33.242,-50.468,179.823,5.876,149.100
C03179=1106.072,-33.492,-50.454,179.823,5.872,149.099
C03180=1106.077,-33.741,-50.442,179.823,5.868,149.099
C03181=1106.082,-33.991,-50.429,179.822,5.863,149.098
C03182=1106.087,-34.241,-50.416,179.822,5.858,149.097
C03183=1106.093,-34.490,-50.403,179.821,5.854,149.096
C03184=1106.098,-34.739,-50.390,179.821,5.850,149.095
C03185=1106.102,-34.989,-50.377,179.821,5.845,149.094
C03186=1106.108,-35.239,-50.364,179.820,5.840,149.093
C03187=1106.113,-35.488,-50.352,179.820,5.836,149.092
C03188=1106.118,-35.738,-50.339,179.820,5.832,149.091
C03189=1106.124,-35.988,-50.325,179.820,5.827,149.091
C03190=1106.129,-36.237,-50.313,179.819,5.822,149.090
C03191=1106.133,-36.487,-50.300,179.819,5.818,149.089
C03192=1106.138,-36.737,-50.287,179.818,5.814,149.088
C03193=1106.143,-36.986,-50.275,179.818,5.809,149.087
C03194=1106.149,-37.236,-50.262,179.817,5.804,149.086
C03195=1106.154,-37.486,-50.249,179.817,5.800,149.085
C03196=1106.159,-37.735,-50.236,179.817,5.795,149.084
C03197=1106.164,-37.984,-50.223,179.817,5.791,149.083
C03198=1106.169,-38.235,-50.210,179.816,5.786,149.083
C03199=1106.174,-38.484,-50.197,179.816,5.782,149.082
C03200=1106.180,-38.733,-50.185,179.815,5.777,149.081
C03201=1106.185,-38.983,-50.172,179.815,5.772,149.080
C03202=1106.189,-39.233,-50.159,179.815,5.767,149.079
C03203=1106.194,-39.482,-50.146,179.815,5.762,149.078
C03204=1106.201,-39.732,-50.134,179.814,5.758,149.077
C03205=1106.206,-39.982,-50.121,179.814,5.754,149.076
C03206=1106.210,-40.232,-50.108,179.814,5.749,149.075
C03207=1106.215,-40.481,-50.096,179.813,5.744,149.074
C03208=1106.220,-40.730,-50.083,179.813,5.739,149.073
C03209=1106.226,-40.979,-50.071,179.813,5.735,149.072
C03210=1106.231,-41.230,-50.058,179.813,5.730,149.071
C03211=1106.236,-41.480,-50.045,179.812,5.725,149.070
C03212=1106.241,-41.729,-50.033,179.812,5.720,149.069
C03213=1106.247,-41.978,-50.020,179.812,5.715,149.068
C03214=1106.252,-42.228,-50.007,179.811,5.709,149.067
C03215=1106.256,-42.478,-49.995,179.810,5.705,149.066
C03216=1106.262,-42.728,-49.982,179.810,5.700,149.065
C03217=1106.267,-42.977,-49.970,179.811,5.696,149.064
C03218=1106.272,-43.226,-49.957,179.811,5.690,149.063
C03219=1106.277,-43.476,-49.945,179.811,5.685,149.062
C03220=1106.282,-43.726,-49.932,179.811,5.681,149.061
C03221=1106.287,-43.976,-49.920,179.811,5.676,149.060
C03222=1106.292,-44.225,-49.907,179.812,5.672,149.059
C03223=1106.298,-44.475,-49.895,179.812,5.667,149.058
C03224=1106.302,-44.689,-49.884,179.812,5.663,149.057
C03225=1106.306,-44.904,-49.873,179.812,5.659,149.056
C03226=1106.310,-45.118,-49.863,179.812,5.655,149.055
C03227=1106.316,-45.332,-49.852,179.812,5.650,149.054
C03228=1106.320,-45.547,-49.842,179.812,5.646,149.053
C03229=1106.324,-45.761,-49.831,179.812,5.642,149.052
C03230=1106.329,-45.975,-49.820,179.812,5.638,149.051
C03231=1106.333,-46.190,-49.809,179.812,5.635,149.050
C03232=1106.338,-46.440,-49.797,179.812,5.629,149.049
C03233=1106.343,-46.689,-49.784,179.813,5.625,149.048
C03234=1106.349,-46.939,-49.772,179.813,5.620,149.047
C03235=1106.354,-47.188,-49.760,179.813,5.615,149.046
C03236=1106.359,-47.437,-49.747,179.813,5.611,149.045
C03237=1106.364,-47.688,-49.735,179.813,5.606,149.044
C03238=1106.369,-47.937,-49.722,179.814,5.602,149.043
C03239=1106.374,-48.187,-49.711,179.814,5.597,149.042
C03240=1106.380,-48.437,-49.698,179.814,5.592,149.040
C03241=1106.385,-48.686,-49.685,179.814,5.588,149.040
C03242=1106.390,-48.936,-49.673,179.814,5.583,149.038
C03243=1106.395,-49.185,-49.661,179.814,5.577,149.037
C03244=1106.400,-49.435,-49.650,179.814,5.573,149.036
C03245=1106.405,-49.684,-49.637,179.814,5.568,149.035
C03246=1106.410,-49.935,-49.625,179.814,5.563,149.034
C03247=1106.415,-50.184,-49.612,179.815,5.559,149.033
C03248=1106.420,-50.434,-49.600,179.815,5.554,149.032
C03249=1106.426,-50.683,-49.588,179.815,5.550,149.031
C03250=1106.431,-50.933,-49.576,179.815,5.545,149.030
C03251=1106.436,-51.183,-49.563,179.815,5.540,149.029
C03252=1106.442,-51.433,-49.551,179.816,5.536,149.028
C03253=1106.447,-51.682,-49.539,179.816,5.530,149.026
C03254=1106.452,-51.932,-49.527,179.815,5.526,149.025
C03255=1106.456,-52.181,-49.515,179.816,5.521,149.024
C03256=1106.462,-52.431,-49.503,179.816,5.516,149.023
C03257=1106.467,-52.680,-49.490,179.816,5.512,149.022
C03258=1106.472,-52.930,-49.478,179.816,5.507,149.021
C03259=1106.478,-53.179,-49.466,179.816,5.502,149.020
C03260=1106.482,-53.430,-49.454,179.816,5.497,149.019
C03261=1106.488,-53.679,-49.441,179.817,5.493,149.018
C03262=1106.492,-53.929,-49.430,179.816,5.488,149.017
C03263=1106.498,-54.179,-49.418,179.816,5.483,149.016
C03264=1106.503,-54.428,-49.405,179.817,5.479,149.015
C03265=1106.508,-54.678,-49.393,179.817,5.474,149.014
C03266=1106.513,-54.927,-49.381,179.817,5.470,149.013
C03267=1106.518,-55.177,-49.369,179.817,5.465,149.011
C03268=1106.523,-55.427,-49.358,179.817,5.460,149.010
C03269=1106.529,-55.676,-49.345,179.818,5.456,149.009
C03270=1106.534,-55.926,-49.333,179.818,5.450,149.008
C03271=1106.539,-56.176,-49.321,179.817,5.446,149.007
C03272=1106.544,-56.425,-49.309,179.818,5.441,149.006
C03273=1106.549,-56.675,-49.297,179.818,5.437,149.005
C03274=1106.555,-56.925,-49.285,179.818,5.431,149.004
C03275=1106.560,-57.174,-49.273,179.818,5.427,149.003
C03276=1106.565,-57.424,-49.261,179.818,5.422,149.002
C03277=1106.570,-57.674,-49.250,179.818,5.417,149.001
C03278=1106.575,-57.923,-49.237,179.818,5.413,149.000
C03279=1106.580,-58.173,-49.225,179.818,5.408,148.999
C03280=1106.585,-58.388,-49.215,179.819,5.404,148.998
C03281=1106.589,-58.602,-49.205,179.819,5.400,148.997
C03282=1106.594,-58.816,-49.195,179.819,5.396,148.996
C03283=1106.598,-59.031,-49.184,179.819,5.392,148.995
C03284=1106.603,-59.245,-49.174,179.819,5.388,148.994
C03285=1106.607,-59.460,-49.164,179.819,5.384,148.993
C03286=1106.611,-59.674,-49.154,179.819,5.380,148.992
C03287=1106.616,-59.888,-49.144,179.819,5.376,148.991
C03288=1106.622,-60.138,-49.132,179.819,5.371,148.990
C03289=1106.626,-60.387,-49.120,179.819,5.366,148.989
C03290=1106.631,-60.637,-49.108,179.818,5.362,148.988
C03291=1106.637,-60.887,-49.096,179.818,5.356,148.987
C03292=1106.641,-61.137,-49.085,179.817,5.351,148.986
C03293=1106.647,-61.386,-49.073,179.817,5.346,148.985
C03294=1106.652,-61.636,-49.061,179.817,5.341,148.984
C03295=1106.657,-61.885,-49.049,179.817,5.336,148.983
C03296=1106.662,-62.135,-49.037,179.817,5.331,148.982
C03297=1106.668,-62.385,-49.026,179.816,5.326,148.981
C03298=1106.672,-62.635,-49.014,179.817,5.321,148.980
C03299=1106.678,-62.885,-49.002,179.816,5.317,148.979
C03300=1106.683,-63.134,-48.991,179.816,5.312,148.978
C03301=1106.688,-63.384,-48.980,179.816,5.307,148.977
C03302=1106.694,-63.633,-48.967,179.816,5.302,148.976
C03303=1106.698,-63.883,-48.956,179.816,5.297,148.975
C03304=1106.704,-64.133,-48.944,179.815,5.292,148.974
C03305=1106.708,-64.382,-48.932,179.815,5.286,148.973
C03306=1106.714,-64.632,-48.921,179.815,5.281,148.972
C03307=1106.719,-64.882,-48.909,179.815,5.276,148.971
C03308=1106.724,-65.131,-48.898,179.815,5.271,148.970
C03309=1106.730,-65.381,-48.886,179.814,5.266,148.969
C03310=1106.735,-65.631,-48.875,179.814,5.261,148.968
C03311=1106.740,-65.881,-48.863,179.815,5.256,148.966
C03312=1106.745,-66.130,-48.851,179.814,5.251,148.965
C03313=1106.750,-66.380,-48.840,179.814,5.246,148.964
C03314=1106.755,-66.629,-48.829,179.814,5.241,148.963
C03315=1106.761,-66.879,-48.817,179.814,5.236,148.962
C03316=1106.766,-67.129,-48.805,179.814,5.231,148.961
C03317=1106.771,-67.378,-48.794,179.814,5.226,148.960
C03318=1106.776,-67.628,-48.782,179.813,5.220,148.959
C03319=1106.781,-67.878,-48.770,179.813,5.215,148.958
C03320=1106.786,-68.127,-48.759,179.814,5.210,148.957
C03321=1106.792,-68.377,-48.748,179.813,5.205,148.956
C03322=1106.797,-68.627,-48.736,179.813,5.200,148.955
C03323=1106.802,-68.877,-48.725,179.813,5.195,148.953
C03324=1106.807,-69.127,-48.714,179.814,5.190,148.952
C03325=1106.813,-69.376,-48.702,179.813,5.185,148.951
C03326=1106.818,-69.626,-48.691,179.813,5.180,148.950
C03327=1106.823,-69.876,-48.679,179.813,5.175,148.949
C03328=1106.828,-70.125,-48.668,179.814,5.170,148.948
C03329=1106.834,-70.374,-48.656,179.814,5.165,148.947
C03330=1106.839,-70.624,-48.645,179.813,5.160,148.946
C03331=1106.844,-70.874,-48.634,179.813,5.155,148.945
C03332=1106.849,-71.124,-48.623,179.814,5.150,148.943
C03333=1106.854,-71.373,-48.612,179.814,5.145,148.942
C03334=1106.860,-71.623,-48.600,179.814,5.139,148.941
C03335=1106.864,-71.873,-48.588,179.814,5.134,148.940
C03336=1106.869,-72.087,-48.579,179.814,5.129,148.939
C03337=1106.874,-72.302,-48.569,179.814,5.126,148.938
C03338=1106.878,-72.517,-48.560,179.814,5.121,148.937
C03339=1106.882,-72.731,-48.550,179.814,5.117,148.936
C03340=1106.887,-72.946,-48.540,179.814,5.112,148.935
C03341=1106.892,-73.160,-48.531,179.814,5.108,148.934
C03342=1106.896,-73.375,-48.521,179.814,5.103,148.933
C03343=1106.900,-73.589,-48.512,179.814,5.099,148.932
C03344=1106.906,-73.839,-48.500,179.814,5.094,148.931
C03345=1106.910,-74.088,-48.489,179.814,5.089,148.930
C03346=1106.916,-74.338,-48.478,179.814,5.084,148.929
C03347=1106.921,-74.588,-48.467,179.815,5.078,148.927
C03348=1106.926,-74.837,-48.455,179.815,5.073,148.926
C03349=1106.932,-75.087,-48.445,179.815,5.068,148.925
C03350=1106.937,-75.337,-48.433,179.815,5.063,148.924
C03351=1106.942,-75.587,-48.422,179.815,5.058,148.923
C03352=1106.947,-75.836,-48.412,179.815,5.053,148.922
C03353=1106.953,-76.086,-48.400,179.815,5.048,148.920
C03354=1106.958,-76.336,-48.388,179.816,5.043,148.919
C03355=1106.963,-76.585,-48.378,179.816,5.037,148.918
C03356=1106.969,-76.835,-48.366,179.816,5.032,148.917
C03357=1106.973,-77.085,-48.355,179.816,5.027,148.916
C03358=1106.979,-77.334,-48.345,179.816,5.022,148.915
C03359=1106.984,-77.584,-48.334,179.816,5.017,148.913
C03360=1106.989,-77.834,-48.322,179.817,5.012,148.912
C03361=1106.995,-78.083,-48.311,179.817,5.007,148.911
C03362=1106.999,-78.333,-48.300,179.817,5.001,148.910
C03363=1107.005,-78.583,-48.290,179.817,4.996,148.909
C03364=1107.010,-78.832,-48.278,179.817,4.991,148.907
C03365=1107.015,-79.083,-48.268,179.817,4.986,148.906
C03366=1107.021,-79.332,-48.257,179.817,4.981,148.905
C03367=1107.026,-79.582,-48.246,179.818,4.976,148.904
C03368=1107.032,-79.831,-48.235,179.818,4.971,148.903
C03369=1107.037,-80.081,-48.224,179.818,4.965,148.901
C03370=1107.041,-80.331,-48.213,179.819,4.960,148.900
C03371=1107.047,-80.581,-48.202,179.819,4.955,148.899
C03372=1107.052,-80.830,-48.191,179.819,4.950,148.898
C03373=1107.058,-81.080,-48.180,179.819,4.944,148.897
C03374=1107.063,-81.330,-48.169,179.819,4.939,148.895
C03375=1107.068,-81.580,-48.158,179.820,4.935,148.894
C03376=1107.073,-81.829,-48.148,179.820,4.930,148.893
C03377=1107.078,-82.079,-48.137,179.820,4.925,148.892
C03378=1107.083,-82.328,-48.126,179.821,4.920,148.891
C03379=1107.088,-82.578,-48.115,179.821,4.914,148.890
C03380=1107.094,-82.827,-48.104,179.821,4.909,148.888
C03381=1107.099,-83.078,-48.093,179.822,4.904,148.887
C03382=1107.104,-83.328,-48.083,179.822,4.899,148.886
C03383=1107.110,-83.577,-48.072,179.822,4.893,148.885
C03384=1107.115,-83.827,-48.061,179.822,4.888,148.883
C03385=1107.120,-84.076,-48.050,179.823,4.884,148.882
C03386=1107.125,-84.326,-48.040,179.823,4.879,148.881
C03387=1107.130,-84.576,-48.030,179.823,4.874,148.880
C03388=1107.136,-84.826,-48.018,179.823,4.869,148.879
C03389=1107.141,-85.075,-48.008,179.824,4.863,148.878
C03390=1107.146,-85.325,-47.996,179.824,4.858,148.876
C03391=1107.152,-85.574,-47.986,179.824,4.853,148.875
C03392=1107.156,-85.790,-47.977,179.825,4.849,148.874
C03393=1107.161,-86.004,-47.968,179.825,4.845,148.873
C03394=1107.164,-86.218,-47.958,179.826,4.840,148.872
C03395=1107.169,-86.433,-47.949,179.825,4.836,148.871
C03396=1107.174,-86.647,-47.940,179.826,4.831,148.870
C03397=1107.178,-86.862,-47.931,179.826,4.827,148.869
C03398=1107.182,-87.076,-47.922,179.826,4.823,148.868
C03399=1107.187,-87.292,-47.913,179.827,4.818,148.867
C03400=1107.193,-87.541,-47.902,179.827,4.813,148.865
C03401=1107.197,-87.791,-47.891,179.828,4.809,148.864
C03402=1107.203,-88.041,-47.881,179.828,4.804,148.863
C03403=1107.208,-88.291,-47.870,179.828,4.799,148.862
C03404=1107.214,-88.540,-47.860,179.828,4.793,148.861
C03405=1107.218,-88.790,-47.849,179.829,4.788,148.859
C03406=1107.224,-89.039,-47.839,179.830,4.784,148.858
C03407=1107.230,-89.289,-47.828,179.830,4.778,148.857
C03408=1107.235,-89.539,-47.818,179.830,4.773,148.856
C03409=1107.240,-89.788,-47.807,179.830,4.768,148.855
C03410=1107.245,-90.038,-47.796,179.831,4.764,148.853
C03411=1107.250,-90.288,-47.786,179.831,4.759,148.852
C03412=1107.255,-90.538,-47.776,179.832,4.753,148.851
C03413=1107.261,-90.788,-47.765,179.832,4.749,148.850
C03414=1107.266,-91.037,-47.754,179.833,4.744,148.849
C03415=1107.271,-91.287,-47.744,179.833,4.739,148.847
C03416=1107.276,-91.537,-47.733,179.833,4.733,148.846
C03417=1107.282,-91.787,-47.723,179.834,4.729,148.845
C03418=1107.287,-92.036,-47.713,179.834,4.724,148.844
C03419=1107.292,-92.287,-47.702,179.835,4.719,148.842
C03420=1107.297,-92.535,-47.692,179.835,4.714,148.841
C03421=1107.302,-92.785,-47.681,179.836,4.709,148.840
C03422=1107.308,-93.035,-47.671,179.836,4.704,148.839
C03423=1107.313,-93.284,-47.661,179.837,4.700,148.838
C03424=1107.318,-93.535,-47.650,179.837,4.695,148.836
C03425=1107.324,-93.784,-47.640,179.838,4.690,148.835
C03426=1107.329,-94.034,-47.630,179.838,4.685,148.834
C03427=1107.334,-94.284,-47.619,179.838,4.680,148.833
C03428=1107.340,-94.533,-47.609,179.839,4.676,148.832
C03429=1107.345,-94.783,-47.598,179.839,4.670,148.831
C03430=1107.350,-95.032,-47.588,179.839,4.665,148.829
C03431=1107.355,-95.283,-47.578,179.839,4.660,148.828
C03432=1107.360,-95.532,-47.568,179.840,4.656,148.827
C03433=1107.366,-95.782,-47.557,179.840,4.651,148.826
C03434=1107.371,-96.032,-47.547,179.841,4.645,148.825
C03435=1107.376,-96.282,-47.537,179.841,4.641,148.823
C03436=1107.382,-96.531,-47.526,179.842,4.636,148.822
C03437=1107.386,-96.781,-47.516,179.842,4.631,148.821
C03438=1107.392,-97.031,-47.506,179.843,4.627,148.820
C03439=1107.397,-97.281,-47.496,179.843,4.621,148.819
C03440=1107.402,-97.530,-47.485,179.843,4.616,148.817
C03441=1107.408,-97.780,-47.475,179.843,4.611,148.816
C03442=1107.413,-98.030,-47.465,179.844,4.607,148.815
C03443=1107.418,-98.279,-47.455,179.844,4.602,148.814
C03444=1107.423,-98.529,-47.445,179.844,4.596,148.813
C03445=1107.428,-98.779,-47.434,179.845,4.592,148.811
C03446=1107.434,-99.029,-47.424,179.845,4.587,148.810
C03447=1107.440,-99.278,-47.414,179.846,4.582,148.809
C03448=1107.444,-99.493,-47.405,179.846,4.578,148.808
C03449=1107.448,-99.708,-47.397,179.847,4.573,148.807
C03450=1107.453,-99.923,-47.388,179.847,4.570,148.806
C03451=1107.458,-100.137,-47.380,179.847,4.565,148.805
C03452=1107.462,-100.352,-47.371,179.848,4.560,148.804
C03453=1107.466,-100.566,-47.362,179.848,4.556,148.803
C03454=1107.471,-100.781,-47.353,179.848,4.552,148.802
C03455=1107.476,-100.995,-47.345,179.848,4.547,148.801
C03456=1107.481,-101.246,-47.334,179.849,4.543,148.799
C03457=1107.486,-101.495,-47.324,179.849,4.538,148.798
C03458=1107.491,-101.745,-47.315,179.850,4.533,148.797
C03459=1107.497,-101.995,-47.305,179.850,4.528,148.796
C03460=1107.502,-102.245,-47.294,179.851,4.523,148.795
C03461=1107.507,-102.494,-47.284,179.851,4.518,148.793
C03462=1107.512,-102.744,-47.274,179.851,4.513,148.792
C03463=1107.517,-102.994,-47.264,179.852,4.509,148.791
C03464=1107.522,-103.243,-47.254,179.852,4.503,148.790
C03465=1107.528,-103.493,-47.245,179.852,4.498,148.789
C03466=1107.534,-103.743,-47.234,179.853,4.493,148.787
C03467=1107.539,-103.993,-47.224,179.853,4.489,148.786
C03468=1107.544,-104.242,-47.214,179.854,4.484,148.785
C03469=1107.549,-104.492,-47.204,179.854,4.478,148.784
C03470=1107.555,-104.742,-47.194,179.854,4.473,148.783
C03471=1107.559,-104.992,-47.184,179.854,4.468,148.781
C03472=1107.565,-105.241,-47.174,179.855,4.464,148.780
C03473=1107.570,-105.491,-47.165,179.855,4.459,148.779
C03474=1107.576,-105.741,-47.155,179.856,4.453,148.778
C03475=1107.581,-105.991,-47.145,179.856,4.448,148.777
C03476=1107.586,-106.240,-47.135,179.857,4.444,148.775
C03477=1107.591,-106.490,-47.125,179.858,4.438,148.774
C03478=1107.597,-106.740,-47.115,179.858,4.433,148.773
C03479=1107.601,-106.990,-47.105,179.858,4.428,148.772
C03480=1107.607,-107.239,-47.095,179.858,4.423,148.770
C03481=1107.612,-107.489,-47.086,179.859,4.419,148.769
C03482=1107.618,-107.739,-47.076,179.859,4.414,148.768
C03483=1107.623,-107.988,-47.066,179.860,4.408,148.767
C03484=1107.628,-108.238,-47.056,179.860,4.403,148.766
C03485=1107.634,-108.489,-47.046,179.861,4.399,148.764
C03486=1107.638,-108.738,-47.037,179.861,4.394,148.763
C03487=1107.644,-108.987,-47.026,179.862,4.388,148.762
C03488=1107.650,-109.237,-47.017,179.862,4.383,148.761
C03489=1107.655,-109.487,-47.007,179.862,4.378,148.759
C03490=1107.660,-109.738,-46.998,179.862,4.373,148.758
C03491=1107.665,-109.987,-46.988,179.863,4.368,148.757
C03492=1107.671,-110.236,-46.978,179.863,4.363,148.756
C03493=1107.676,-110.486,-46.969,179.864,4.358,148.755
C03494=1107.681,-110.736,-46.959,179.864,4.353,148.753
C03495=1107.686,-110.985,-46.949,179.864,4.348,148.752
C03496=1107.692,-111.236,-46.939,179.866,4.343,148.751
C03497=1107.696,-111.485,-46.930,179.866,4.338,148.749
C03498=1107.702,-111.735,-46.920,179.866,4.333,148.748
C03499=1107.708,-111.985,-46.910,179.866,4.328,148.747
C03500=1107.713,-112.235,-46.901,179.867,4.322,148.746
C03501=1107.719,-112.484,-46.891,179.867,4.317,148.745
C03502=1107.724,-112.734,-46.882,179.867,4.312,148.743
C03503=1107.729,-112.984,-46.871,179.868,4.307,148.742
C03504=1107.733,-113.199,-46.863,179.868,4.303,148.741
C03505=1107.738,-113.413,-46.855,179.869,4.298,148.740
C03506=1107.743,-113.628,-46.847,179.869,4.294,148.739
C03507=1107.747,-113.843,-46.839,179.869,4.290,148.738
C03508=1107.752,-114.057,-46.830,179.870,4.285,148.737
C03509=1107.756,-114.272,-46.822,179.870,4.281,148.736
C03510=1107.760,-114.487,-46.814,179.871,4.276,148.734
C03511=1107.765,-114.702,-46.806,179.871,4.272,148.733
C03512=1107.771,-114.952,-46.796,179.871,4.267,148.732
C03513=1107.776,-115.201,-46.787,179.872,4.261,148.731
C03514=1107.781,-115.451,-46.778,179.872,4.256,148.730
C03515=1107.786,-115.701,-46.767,179.873,4.252,148.728
C03516=1107.792,-115.951,-46.759,179.873,4.247,148.727
C03517=1107.797,-116.200,-46.748,179.874,4.241,148.726
C03518=1107.802,-116.450,-46.739,179.874,4.236,148.725
C03519=1107.808,-116.700,-46.729,179.875,4.231,148.723
C03520=1107.813,-116.949,-46.720,179.875,4.226,148.722
C03521=1107.818,-117.199,-46.711,179.875,4.221,148.721
C03522=1107.824,-117.449,-46.701,179.876,4.215,148.719
C03523=1107.829,-117.699,-46.692,179.876,4.210,148.718
C03524=1107.834,-117.949,-46.682,179.876,4.205,148.717
C03525=1107.839,-118.199,-46.673,179.877,4.199,148.716
C03526=1107.844,-118.449,-46.664,179.878,4.195,148.714
C03527=1107.850,-118.698,-46.654,179.878,4.190,148.713
C03528=1107.855,-118.948,-46.645,179.879,4.184,148.712
C03529=1107.860,-119.198,-46.636,179.879,4.179,148.710
C03530=1107.866,-119.447,-46.626,179.880,4.174,148.709
C03531=1107.871,-119.697,-46.617,179.880,4.169,148.708
C03532=1107.876,-119.947,-46.608,179.881,4.163,148.707
C03533=1107.882,-120.197,-46.598,179.881,4.158,148.705
C03534=1107.887,-120.446,-46.589,179.881,4.153,148.704
C03535=1107.892,-120.696,-46.580,179.882,4.148,148.703
C03536=1107.898,-120.946,-46.570,179.882,4.142,148.701
C03537=1107.903,-121.196,-46.561,179.883,4.137,148.700
C03538=1107.908,-121.446,-46.552,179.883,4.132,148.699
C03539=1107.914,-121.696,-46.542,179.884,4.126,148.698
C03540=1107.919,-121.945,-46.533,179.884,4.121,148.696
C03541=1107.924,-122.195,-46.524,179.884,4.116,148.695
C03542=1107.929,-122.445,-46.515,179.885,4.110,148.694
C03543=1107.935,-122.695,-46.506,179.886,4.105,148.692
C03544=1107.940,-122.944,-46.496,179.886,4.100,148.691
C03545=1107.945,-123.194,-46.487,179.887,4.094,148.690
C03546=1107.951,-123.444,-46.478,179.887,4.089,148.689
C03547=1107.956,-123.694,-46.469,179.888,4.084,148.687
C03548=1107.961,-123.943,-46.459,179.888,4.079,148.686
C03549=1107.966,-124.193,-46.450,179.889,4.073,148.684
C03550=1107.972,-124.443,-46.441,179.889,4.068,148.683
C03551=1107.978,-124.692,-46.432,179.889,4.063,148.682
C03552=1107.983,-124.942,-46.423,179.890,4.057,148.680
C03553=1107.988,-125.192,-46.414,179.891,4.052,148.679
C03554=1107.993,-125.441,-46.405,179.891,4.047,148.678
C03555=1107.999,-125.691,-46.395,179.892,4.041,148.677
C03556=1108.004,-125.941,-46.386,179.892,4.036,148.675
C03557=1108.009,-126.191,-46.377,179.893,4.031,148.674
C03558=1108.014,-126.441,-46.369,179.893,4.026,148.673
C03559=1108.020,-126.691,-46.360,179.894,4.020,148.671
C03560=1108.024,-126.905,-46.351,179.895,4.016,148.670
C03561=1108.029,-127.120,-46.344,179.895,4.011,148.669
C03562=1108.034,-127.335,-46.336,179.895,4.006,148.668
C03563=1108.038,-127.550,-46.328,179.896,4.001,148.667
C03564=1108.043,-127.765,-46.320,179.897,3.997,148.665
C03565=1108.047,-127.980,-46.313,179.896,3.992,148.664
C03566=1108.052,-128.194,-46.305,179.897,3.988,148.663
C03567=1108.056,-128.409,-46.297,179.898,3.983,148.662
C03568=1107.634,-128.399,-46.323,179.905,3.987,148.661
C03569=1107.629,-128.185,-46.331,179.904,3.991,148.662
C03570=1107.624,-127.970,-46.339,179.904,3.996,148.663
C03571=1107.620,-127.755,-46.347,179.903,4.001,148.664
C03572=1107.616,-127.541,-46.354,179.903,4.006,148.665
C03573=1107.611,-127.326,-46.362,179.903,4.010,148.666
C03574=1107.606,-127.111,-46.370,179.902,4.015,148.667
C03575=1107.601,-126.896,-46.378,179.901,4.019,148.669
C03576=1107.597,-126.681,-46.385,179.901,4.025,148.670
C03577=1107.592,-126.432,-46.395,179.901,4.030,148.671
C03578=1107.587,-126.182,-46.404,179.900,4.035,148.673
C03579=1107.581,-125.932,-46.413,179.900,4.040,148.674
C03580=1107.576,-125.682,-46.422,179.899,4.046,148.675
C03581=1107.570,-125.432,-46.431,179.899,4.051,148.677
C03582=1107.565,-125.182,-46.440,179.898,4.056,148.678
C03583=1107.560,-124.934,-46.449,179.897,4.062,148.679
C03584=1107.554,-124.683,-46.459,179.897,4.067,148.680
C03585=1107.549,-124.434,-46.468,179.896,4.073,148.682
C03586=1107.544,-124.184,-46.476,179.896,4.078,148.683
C03587=1107.538,-123.934,-46.485,179.895,4.083,148.685
C03588=1107.533,-123.684,-46.496,179.895,4.088,148.686
C03589=1107.528,-123.435,-46.504,179.895,4.094,148.687
C03590=1107.522,-123.185,-46.513,179.894,4.099,148.688
C03591=1107.517,-122.935,-46.522,179.894,4.104,148.690
C03592=1107.512,-122.685,-46.532,179.893,4.109,148.691
C03593=1107.507,-122.435,-46.541,179.892,4.115,148.692
C03594=1107.501,-122.186,-46.550,179.892,4.120,148.694
C03595=1107.496,-121.936,-46.560,179.891,4.126,148.695
C03596=1107.491,-121.686,-46.569,179.891,4.131,148.696
C03597=1107.485,-121.436,-46.578,179.891,4.136,148.698
C03598=1107.480,-121.186,-46.588,179.890,4.142,148.699
C03599=1107.475,-120.937,-46.597,179.890,4.147,148.700
C03600=1107.469,-120.687,-46.606,179.889,4.152,148.701
C03601=1107.464,-120.437,-46.616,179.888,4.157,148.703
C03602=1107.459,-120.188,-46.625,179.888,4.162,148.704
C03603=1107.454,-119.938,-46.634,179.887,4.167,148.705
C03604=1107.448,-119.688,-46.644,179.887,4.172,148.707
C03605=1107.443,-119.438,-46.653,179.886,4.178,148.708
C03606=1107.438,-119.188,-46.663,179.886,4.183,148.709
C03607=1107.433,-118.938,-46.673,179.886,4.188,148.710
C03608=1107.427,-118.688,-46.682,179.885,4.193,148.712
C03609=1107.422,-118.439,-46.691,179.885,4.199,148.713
C03610=1107.417,-118.189,-46.701,179.884,4.204,148.714
C03611=1107.412,-117.939,-46.710,179.884,4.209,148.716
C03612=1107.406,-117.689,-46.719,179.883,4.214,148.717
C03613=1107.401,-117.440,-46.729,179.883,4.220,148.718
C03614=1107.395,-117.190,-46.738,179.882,4.224,148.719
C03615=1107.390,-116.940,-46.748,179.882,4.230,148.721
C03616=1107.385,-116.691,-46.757,179.881,4.235,148.722
C03617=1107.379,-116.441,-46.767,179.881,4.240,148.723
C03618=1107.374,-116.191,-46.776,179.881,4.245,148.724
C03619=1107.368,-115.942,-46.786,179.880,4.251,148.726
C03620=1107.363,-115.692,-46.795,179.880,4.256,148.727
C03621=1107.358,-115.442,-46.806,179.879,4.261,148.728
C03622=1107.353,-115.192,-46.815,179.879,4.266,148.730
C03623=1107.348,-114.942,-46.825,179.878,4.270,148.731
C03624=1107.342,-114.692,-46.834,179.877,4.276,148.732
C03625=1107.338,-114.478,-46.842,179.878,4.281,148.733
C03626=1107.333,-114.263,-46.850,179.877,4.285,148.734
C03627=1107.329,-114.048,-46.858,179.877,4.289,148.735
C03628=1107.324,-113.834,-46.866,179.877,4.294,148.736
C03629=1107.320,-113.619,-46.875,179.876,4.298,148.738
C03630=1107.316,-113.404,-46.883,179.876,4.302,148.739
C03631=1107.310,-113.189,-46.891,179.875,4.307,148.740
C03632=1107.306,-112.974,-46.900,179.875,4.311,148.741
C03633=1107.301,-112.725,-46.909,179.875,4.316,148.742
C03634=1107.295,-112.475,-46.919,179.874,4.322,148.743
C03635=1107.290,-112.226,-46.929,179.873,4.326,148.745
C03636=1107.284,-111.976,-46.939,179.873,4.331,148.746
C03637=1107.280,-111.726,-46.948,179.873,4.337,148.747
C03638=1107.274,-111.476,-46.958,179.872,4.342,148.748
C03639=1107.269,-111.226,-46.967,179.872,4.347,148.749
C03640=1107.263,-110.977,-46.977,179.871,4.352,148.751
C03641=1107.259,-110.727,-46.987,179.871,4.357,148.752
C03642=1107.253,-110.477,-46.996,179.870,4.362,148.753
C03643=1107.248,-110.227,-47.007,179.870,4.367,148.754
C03644=1107.243,-109.978,-47.017,179.870,4.372,148.756
C03645=1107.237,-109.728,-47.026,179.870,4.377,148.757
C03646=1107.232,-109.478,-47.036,179.869,4.382,148.758
C03647=1107.226,-109.228,-47.045,179.868,4.387,148.759
C03648=1107.222,-108.978,-47.055,179.868,4.392,148.761
C03649=1107.216,-108.729,-47.065,179.867,4.398,148.762
C03650=1107.211,-108.479,-47.076,179.867,4.403,148.763
C03651=1107.206,-108.229,-47.085,179.866,4.407,148.764
C03652=1107.200,-107.980,-47.095,179.866,4.412,148.766
C03653=1107.196,-107.730,-47.105,179.866,4.417,148.767
C03654=1107.190,-107.480,-47.114,179.866,4.422,148.768
C03655=1107.184,-107.230,-47.124,179.865,4.428,148.769
C03656=1107.179,-106.981,-47.134,179.865,4.432,148.770
C03657=1107.174,-106.731,-47.144,179.864,4.437,148.772
C03658=1107.168,-106.481,-47.154,179.864,4.442,148.773
C03659=1107.164,-106.231,-47.164,179.864,4.447,148.774
C03660=1107.158,-105.982,-47.174,179.863,4.452,148.775
C03661=1107.152,-105.732,-47.184,179.862,4.457,148.777
C03662=1107.148,-105.482,-47.193,179.862,4.462,148.778
C03663=1107.142,-105.232,-47.204,179.862,4.468,148.779
C03664=1107.137,-104.983,-47.213,179.862,4.473,148.780
C03665=1107.132,-104.733,-47.223,179.861,4.477,148.781
C03666=1107.127,-104.483,-47.234,179.861,4.482,148.783
C03667=1107.121,-104.233,-47.243,179.860,4.487,148.784
C03668=1107.116,-103.984,-47.253,179.860,4.493,148.785
C03669=1107.110,-103.734,-47.263,179.859,4.497,148.786
C03670=1107.105,-103.484,-47.274,179.859,4.502,148.787
C03671=1107.100,-103.235,-47.283,179.859,4.507,148.789
C03672=1107.095,-102.985,-47.294,179.859,4.512,148.790
C03673=1107.090,-102.735,-47.304,179.858,4.517,148.791
C03674=1107.085,-102.485,-47.313,179.858,4.522,148.792
C03675=1107.079,-102.235,-47.323,179.857,4.527,148.793
C03676=1107.074,-101.985,-47.334,179.857,4.532,148.795
C03677=1107.069,-101.736,-47.344,179.856,4.536,148.796
C03678=1107.064,-101.486,-47.354,179.856,4.542,148.797
C03679=1107.058,-101.237,-47.364,179.856,4.547,148.798
C03680=1107.053,-100.987,-47.375,179.855,4.551,148.799
C03681=1107.049,-100.772,-47.383,179.855,4.556,148.801
C03682=1107.043,-100.557,-47.392,179.855,4.560,148.802
C03683=1107.039,-100.342,-47.400,179.854,4.564,148.803
C03684=1107.035,-100.128,-47.409,179.853,4.569,148.804
C03685=1107.031,-99.914,-47.418,179.853,4.572,148.805
C03686=1107.025,-99.699,-47.427,179.853,4.577,148.806
C03687=1107.022,-99.484,-47.435,179.853,4.582,148.807
C03688=1107.017,-99.270,-47.444,179.852,4.586,148.808
C03689=1107.011,-99.020,-47.454,179.852,4.591,148.809
C03690=1107.006,-98.770,-47.464,179.852,4.596,148.810
C03691=1107.001,-98.520,-47.475,179.851,4.600,148.811
C03692=1106.995,-98.271,-47.485,179.851,4.605,148.813
C03693=1106.990,-98.020,-47.496,179.851,4.610,148.814
C03694=1106.985,-97.771,-47.505,179.850,4.615,148.815
C03695=1106.980,-97.522,-47.515,179.850,4.620,148.816
C03696=1106.975,-97.271,-47.526,179.849,4.625,148.817
C03697=1106.969,-97.022,-47.536,179.849,4.629,148.819
C03698=1106.964,-96.772,-47.546,179.848,4.635,148.820
C03699=1106.959,-96.522,-47.557,179.848,4.640,148.821
C03700=1106.954,-96.273,-47.567,179.848,4.645,148.822
